% RSLogix 500 project C8011 TOPCOAT A 20170522 CBP.RSS, saved by version 8.30.00.16 %
PROJECT "C8011"    % processor: MicroLogix 1400; MAIN_PROG %

PROGRAM FILES
  LAD 2 "MAIN_PROG"  16 rungs
  LAD 3 "XFR 4"  40 rungs
  LAD 4 "XFR 5"  10 rungs
  LAD 5 "XFR 6"  10 rungs
  LAD 6 "XFR 7"  24 rungs
  LAD 7 "XFR 8"  19 rungs
  LAD 8 "XFR 9"  16 rungs
  LAD 9 "XFR 10"  27 rungs
  LAD 10 "XFR 14"  3 rungs
  LAD 11 "RFID SB"  8 rungs
  LAD 12 "Z24_Z21"  10 rungs
  LAD 13 "Z90_Z92"  4 rungs
  LAD 14 "Z49_Z54"  1 rungs
  LAD 15 "COMM"  19 rungs
  LAD 16 "XFR 69"  14 rungs

DATA FILES
  O0 OUTPUT  10 elements
  I1 INPUT  11 elements
  S2 STATUS  66 elements
  B3 BINARY  20 elements
  T4 TIMER  100 elements
  C5 COUNTER  20 elements
  R6 CONTROL  10 elements
  N7 INTEGER  100 elements
  F8 FLOAT  1 elements
  MG9   10 elements
  RI10   10 elements
  ST12 MATERIALS  50 elements
  ST13 RFID DATA  2 elements

LADDER 2 "MAIN_PROG"
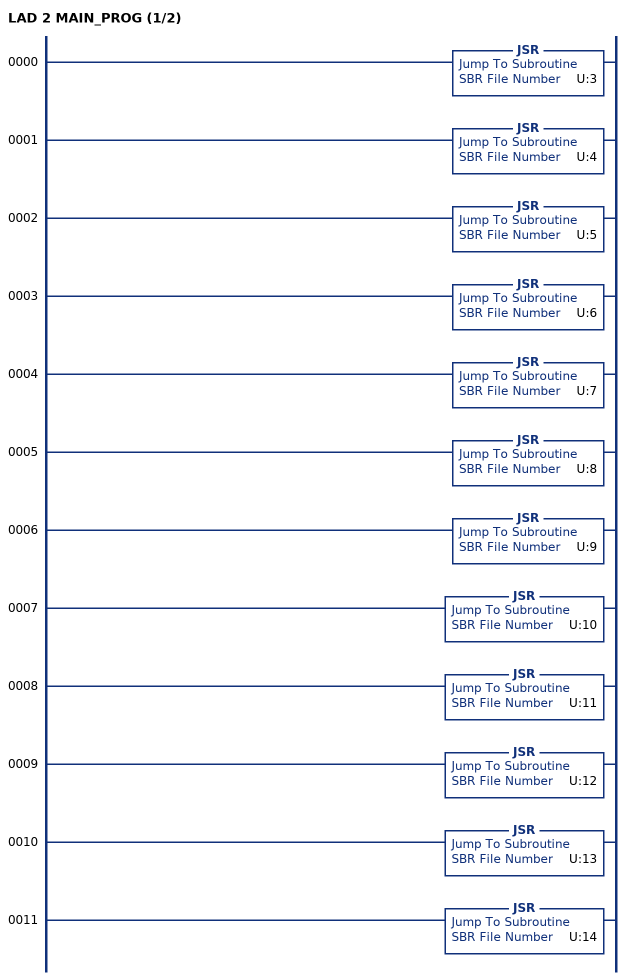
% Rung: 0 %
SOR JSR U:3 EOR
% Rung: 1 %
SOR JSR U:4 EOR
% Rung: 2 %
SOR JSR U:5 EOR
% Rung: 3 %
SOR JSR U:6 EOR
% Rung: 4 %
SOR JSR U:7 EOR
% Rung: 5 %
SOR JSR U:8 EOR
% Rung: 6 %
SOR JSR U:9 EOR
% Rung: 7 %
SOR JSR U:10 EOR
% Rung: 8 %
SOR JSR U:11 EOR
% Rung: 9 %
SOR JSR U:12 EOR
% Rung: 10 %
SOR JSR U:13 EOR
% Rung: 11 %
SOR JSR U:14 EOR

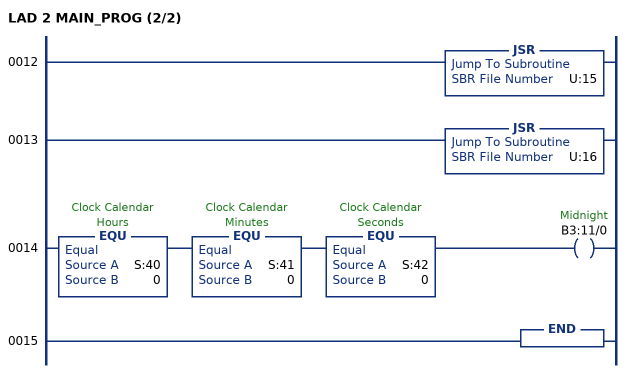
% Rung: 12 %
SOR JSR U:15 EOR
% Rung: 13 %
SOR JSR U:16 EOR
% Rung: 14 %
SOR EQU S:40 0 EQU S:41 0 EQU S:42 0 OTE B3:11/0 EOR
%   S:40  "Clock Calendar Hours" %
%   S:41  "Clock Calendar Minutes" %
%   S:42  "Clock Calendar Seconds" %
%   B3:11/0  "Midnight" %
% Rung: 15 %
SOR END EOR

LADDER 3 "XFR 4"
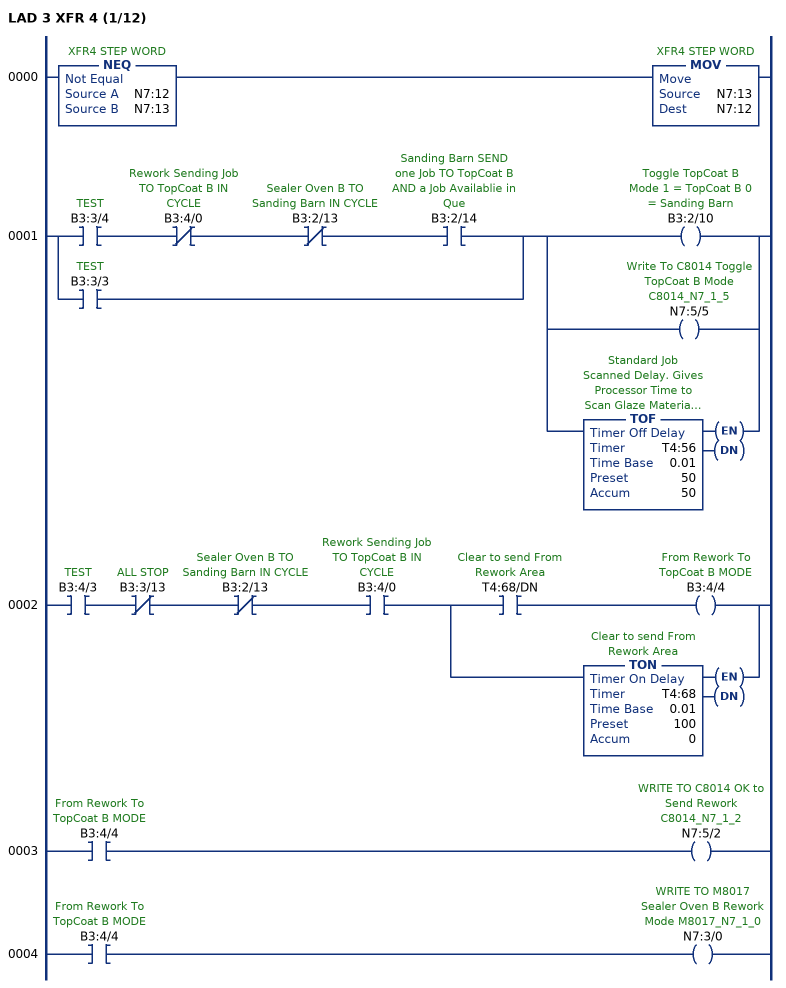
% Rung: 0 %
SOR NEQ N7:12 N7:13 MOV N7:13 N7:12 EOR
%   N7:12  "XFR4 STEP WORD" %
% Rung: 1 %
SOR BST XIC B3:3/4 XIO B3:4/0 XIO B3:2/13 XIC B3:2/14 NXB XIC B3:3/3 BND BST OTE B3:2/10 NXB OTE N7:5/5 NXB TOF T4:56 0.01 50 50 BND EOR
%   B3:3/4  "TEST" %
%   B3:4/0  "Rework Sending Job TO TopCoat B IN CYCLE" %
%   B3:2/13  "Sealer Oven B TO Sanding Barn IN CYCLE" %
%   B3:2/14  "Sanding Barn SEND one Job TO TopCoat B AND a Job Availablie in Que" %
%   B3:3/3  "TEST" %
%   B3:2/10  "Toggle TopCoat B Mode 1 = TopCoat B 0 = Sanding Barn" %
%   N7:5/5  C8014_N7_1_5  "Write To C8014 Toggle TopCoat B Mode" %
%   T4:56  "Standard Job Scanned Delay. Gives Processor Time to Scan Glaze Material Numbers" %
% Rung: 2 %
SOR XIC B3:4/3 XIO B3:3/13 XIO B3:2/13 XIC B3:4/0 BST XIC T4:68/DN OTE B3:4/4 NXB TON T4:68 0.01 100 0 BND EOR
%   B3:4/3  "TEST" %
%   B3:3/13  "ALL STOP" %
%   B3:2/13  "Sealer Oven B TO Sanding Barn IN CYCLE" %
%   B3:4/0  "Rework Sending Job TO TopCoat B IN CYCLE" %
%   T4:68  "Clear to send From Rework Area" %
%   B3:4/4  "From Rework To TopCoat B MODE" %
% Rung: 3 %
SOR XIC B3:4/4 OTE N7:5/2 EOR
%   B3:4/4  "From Rework To TopCoat B MODE" %
%   N7:5/2  C8014_N7_1_2  "WRITE TO C8014 OK to Send Rework" %
% Rung: 4 %
SOR XIC B3:4/4 OTE N7:3/0 EOR
%   B3:4/4  "From Rework To TopCoat B MODE" %
%   N7:3/0  M8017_N7_1_0  "WRITE TO M8017 Sealer Oven B Rework Mode" %

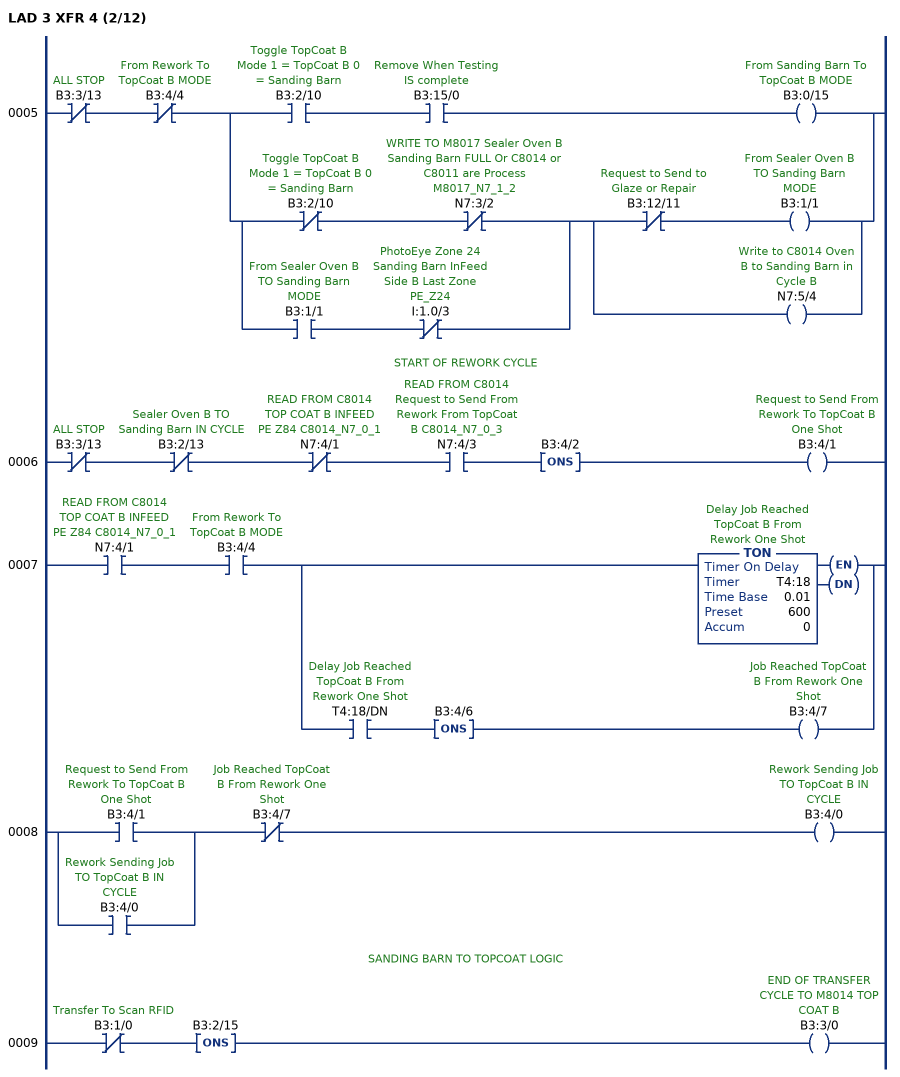
% Rung: 5 %
SOR XIO B3:3/13 XIO B3:4/4 BST XIC B3:2/10 XIC B3:15/0 OTE B3:0/15 NXB BST XIO B3:2/10 XIO N7:3/2 NXB XIC B3:1/1 XIO I:1.0/3 BND BST XIO B3:12/11 OTE B3:1/1 NXB OTE N7:5/4 BND BND EOR
%   B3:3/13  "ALL STOP" %
%   B3:4/4  "From Rework To TopCoat B MODE" %
%   B3:2/10  "Toggle TopCoat B Mode 1 = TopCoat B 0 = Sanding Barn" %
%   B3:15/0  "Remove When Testing IS complete" %
%   B3:0/15  "From Sanding Barn To TopCoat B MODE" %
%   N7:3/2  M8017_N7_1_2  "WRITE TO M8017 Sealer Oven B Sanding Barn FULL Or C8014 or C8011 are Process" %
%   B3:1/1  "From Sealer Oven B TO Sanding Barn MODE" %
%   I:1.0/3  PE_Z24  "PhotoEye Zone 24 Sanding Barn InFeed Side B Last Zone" %
%   B3:12/11  "Request to Send to Glaze or Repair" %
%   N7:5/4  B  "Write to C8014 Oven B to Sanding Barn in Cycle" %
% Rung: 6 %
% START OF REWORK CYCLE %
SOR XIO B3:3/13 XIO B3:2/13 XIO N7:4/1 XIC N7:4/3 ONS B3:4/2 OTE B3:4/1 EOR
%   B3:3/13  "ALL STOP" %
%   B3:2/13  "Sealer Oven B TO Sanding Barn IN CYCLE" %
%   N7:4/1  C8014_N7_0_1  "READ FROM C8014 TOP COAT B INFEED PE Z84" %
%   N7:4/3  C8014_N7_0_3  "READ FROM C8014 Request to Send From Rework From TopCoat B" %
%   B3:4/1  "Request to Send From Rework To TopCoat B One Shot" %
% Rung: 7 %
SOR XIC N7:4/1 XIC B3:4/4 BST TON T4:18 0.01 600 0 NXB XIC T4:18/DN ONS B3:4/6 OTE B3:4/7 BND EOR
%   N7:4/1  C8014_N7_0_1  "READ FROM C8014 TOP COAT B INFEED PE Z84" %
%   B3:4/4  "From Rework To TopCoat B MODE" %
%   T4:18  "Delay Job Reached TopCoat B From Rework One Shot" %
%   B3:4/7  "Job Reached TopCoat B From Rework One Shot" %
% Rung: 8 %
SOR BST XIC B3:4/1 NXB XIC B3:4/0 BND XIO B3:4/7 OTE B3:4/0 EOR
%   B3:4/1  "Request to Send From Rework To TopCoat B One Shot" %
%   B3:4/0  "Rework Sending Job TO TopCoat B IN CYCLE" %
%   B3:4/7  "Job Reached TopCoat B From Rework One Shot" %
% Rung: 9 %
% SANDING BARN TO TOPCOAT LOGIC %
SOR XIO B3:1/0 ONS B3:2/15 OTE B3:3/0 EOR
%   B3:1/0  "Transfer To Scan RFID" %
%   B3:3/0  "END OF TRANSFER CYCLE TO M8014 TOP COAT B" %

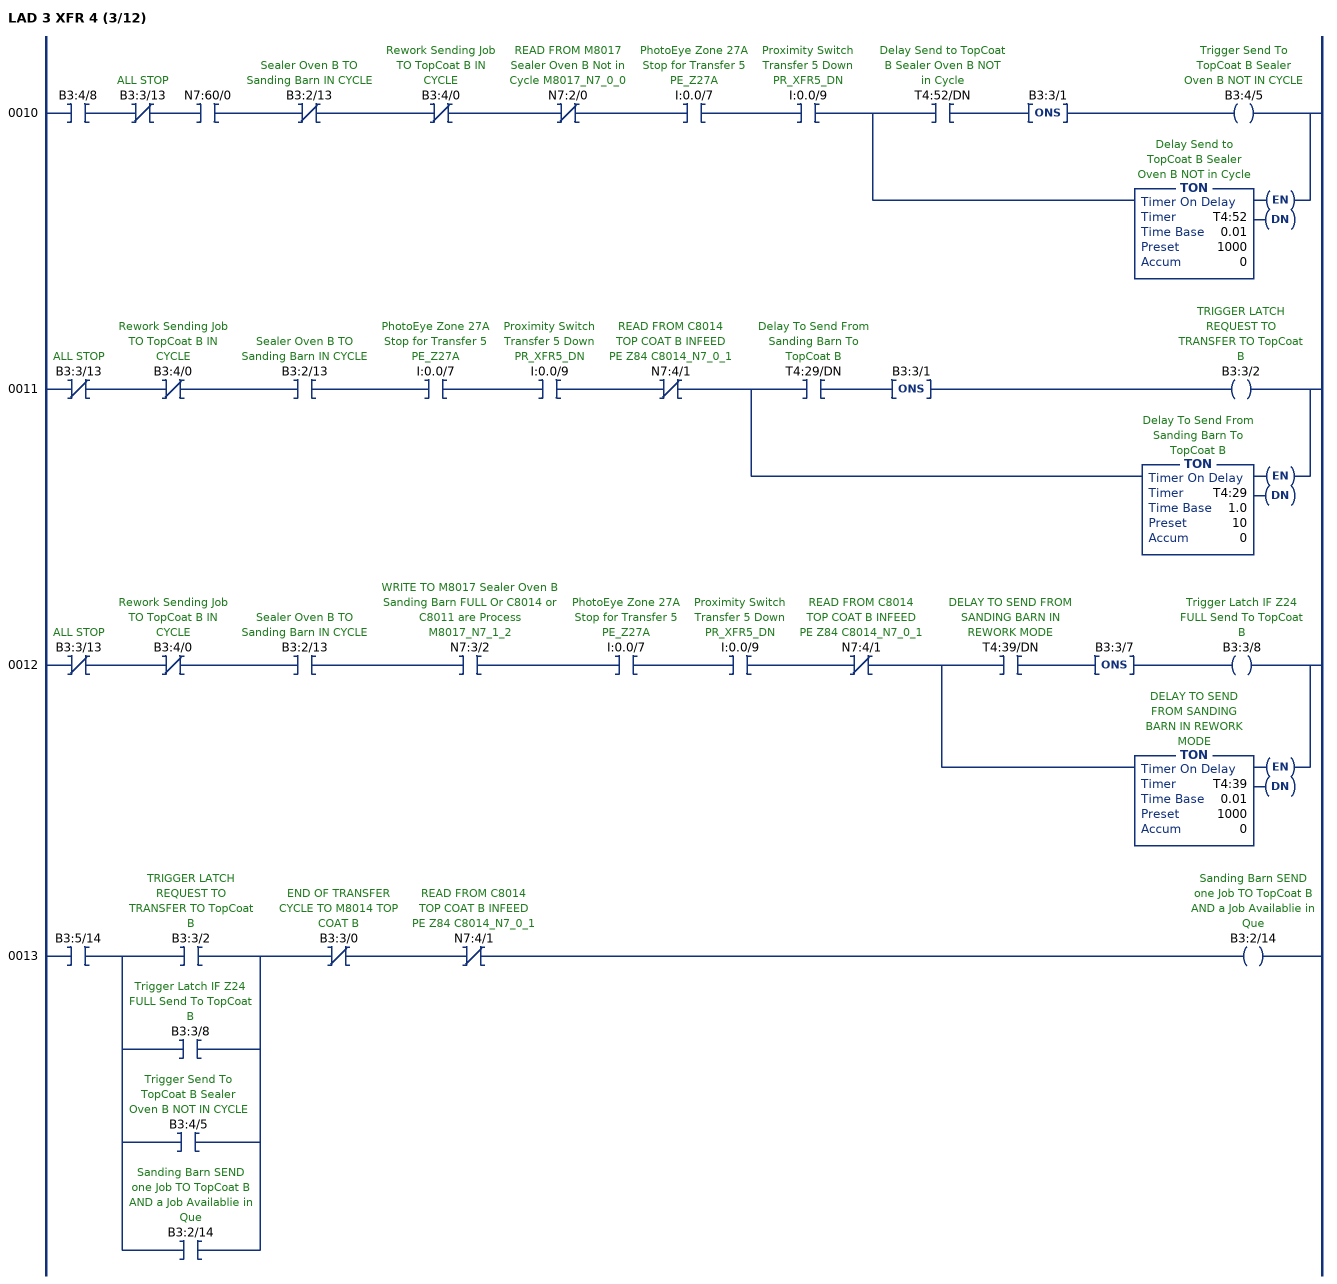
% Rung: 10 %
SOR XIC B3:4/8 XIO B3:3/13 XIC N7:60/0 XIO B3:2/13 XIO B3:4/0 XIO N7:2/0 XIC I:0.0/7 XIC I:0.0/9 BST XIC T4:52/DN ONS B3:3/1 OTE B3:4/5 NXB TON T4:52 0.01 1000 0 BND EOR
%   B3:3/13  "ALL STOP" %
%   B3:2/13  "Sealer Oven B TO Sanding Barn IN CYCLE" %
%   B3:4/0  "Rework Sending Job TO TopCoat B IN CYCLE" %
%   N7:2/0  M8017_N7_0_0  "READ FROM M8017 Sealer Oven B Not in Cycle" %
%   I:0.0/7  PE_Z27A  "PhotoEye Zone 27A Stop for Transfer 5" %
%   I:0.0/9  PR_XFR5_DN  "Proximity Switch Transfer 5 Down" %
%   T4:52  "Delay Send to TopCoat B Sealer Oven B NOT in Cycle" %
%   B3:4/5  "Trigger Send To TopCoat B Sealer Oven B NOT IN CYCLE" %
% Rung: 11 %
SOR XIO B3:3/13 XIO B3:4/0 XIC B3:2/13 XIC I:0.0/7 XIC I:0.0/9 XIO N7:4/1 BST XIC T4:29/DN ONS B3:3/1 OTE B3:3/2 NXB TON T4:29 1.0 10 0 BND EOR
%   B3:3/13  "ALL STOP" %
%   B3:4/0  "Rework Sending Job TO TopCoat B IN CYCLE" %
%   B3:2/13  "Sealer Oven B TO Sanding Barn IN CYCLE" %
%   I:0.0/7  PE_Z27A  "PhotoEye Zone 27A Stop for Transfer 5" %
%   I:0.0/9  PR_XFR5_DN  "Proximity Switch Transfer 5 Down" %
%   N7:4/1  C8014_N7_0_1  "READ FROM C8014 TOP COAT B INFEED PE Z84" %
%   T4:29  "Delay To Send From Sanding Barn To TopCoat B" %
%   B3:3/2  "TRIGGER LATCH REQUEST TO TRANSFER TO TopCoat B" %
% Rung: 12 %
SOR XIO B3:3/13 XIO B3:4/0 XIC B3:2/13 XIC N7:3/2 XIC I:0.0/7 XIC I:0.0/9 XIO N7:4/1 BST XIC T4:39/DN ONS B3:3/7 OTE B3:3/8 NXB TON T4:39 0.01 1000 0 BND EOR
%   B3:3/13  "ALL STOP" %
%   B3:4/0  "Rework Sending Job TO TopCoat B IN CYCLE" %
%   B3:2/13  "Sealer Oven B TO Sanding Barn IN CYCLE" %
%   N7:3/2  M8017_N7_1_2  "WRITE TO M8017 Sealer Oven B Sanding Barn FULL Or C8014 or C8011 are Process" %
%   I:0.0/7  PE_Z27A  "PhotoEye Zone 27A Stop for Transfer 5" %
%   I:0.0/9  PR_XFR5_DN  "Proximity Switch Transfer 5 Down" %
%   N7:4/1  C8014_N7_0_1  "READ FROM C8014 TOP COAT B INFEED PE Z84" %
%   T4:39  "DELAY TO SEND FROM SANDING BARN IN REWORK MODE" %
%   B3:3/8  "Trigger Latch IF Z24 FULL Send To TopCoat B" %
% Rung: 13 %
SOR XIC B3:5/14 BST XIC B3:3/2 NXB XIC B3:3/8 NXB XIC B3:4/5 NXB XIC B3:2/14 BND XIO B3:3/0 XIO N7:4/1 OTE B3:2/14 EOR
%   B3:3/2  "TRIGGER LATCH REQUEST TO TRANSFER TO TopCoat B" %
%   B3:3/8  "Trigger Latch IF Z24 FULL Send To TopCoat B" %
%   B3:4/5  "Trigger Send To TopCoat B Sealer Oven B NOT IN CYCLE" %
%   B3:2/14  "Sanding Barn SEND one Job TO TopCoat B AND a Job Availablie in Que" %
%   B3:3/0  "END OF TRANSFER CYCLE TO M8014 TOP COAT B" %
%   N7:4/1  C8014_N7_0_1  "READ FROM C8014 TOP COAT B INFEED PE Z84" %

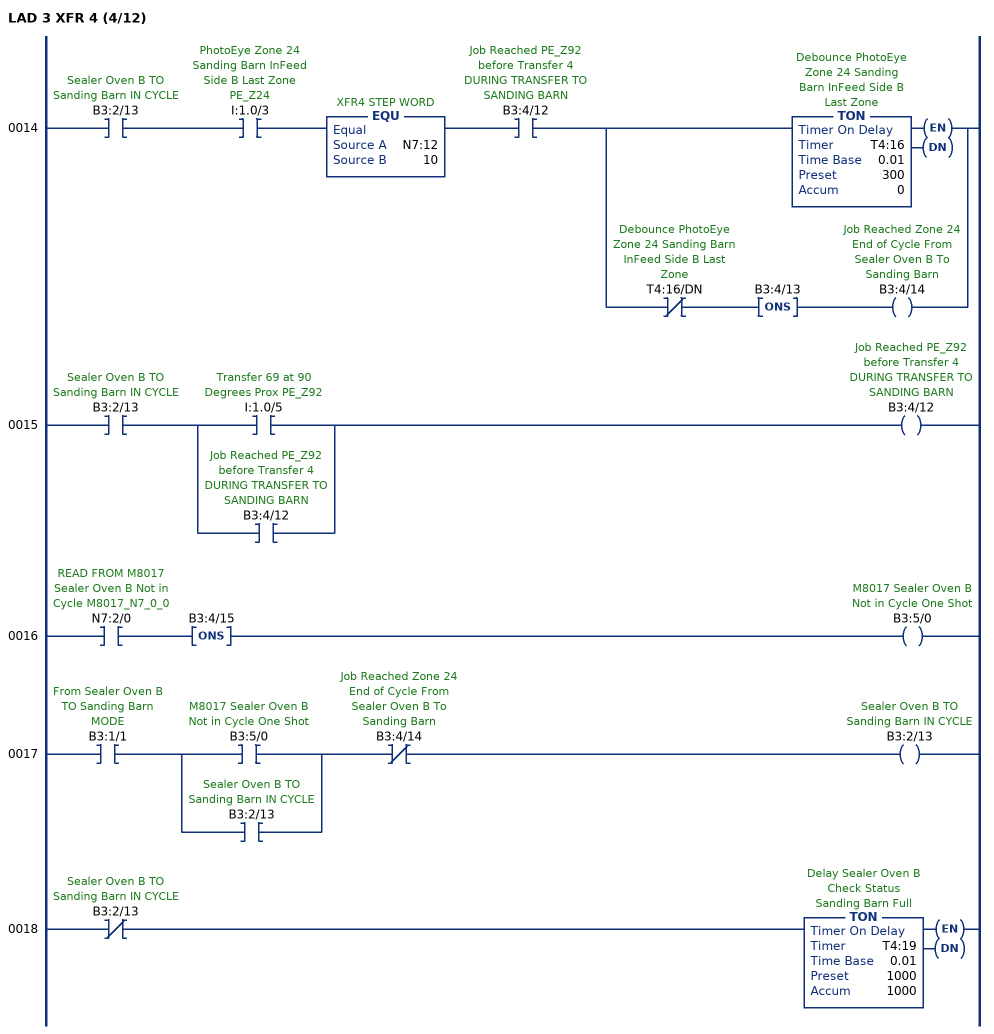
% Rung: 14 %
SOR XIC B3:2/13 XIC I:1.0/3 EQU N7:12 10 XIC B3:4/12 BST TON T4:16 0.01 300 0 NXB XIO T4:16/DN ONS B3:4/13 OTE B3:4/14 BND EOR
%   B3:2/13  "Sealer Oven B TO Sanding Barn IN CYCLE" %
%   I:1.0/3  PE_Z24  "PhotoEye Zone 24 Sanding Barn InFeed Side B Last Zone" %
%   N7:12  "XFR4 STEP WORD" %
%   B3:4/12  "Job Reached PE_Z92 before Transfer 4 DURING TRANSFER TO SANDING BARN" %
%   T4:16  "Debounce PhotoEye Zone 24 Sanding Barn InFeed Side B Last Zone" %
%   B3:4/14  "Job Reached Zone 24 End of Cycle From Sealer Oven B To Sanding Barn" %
% Rung: 15 %
SOR XIC B3:2/13 BST XIC I:1.0/5 NXB XIC B3:4/12 BND OTE B3:4/12 EOR
%   B3:2/13  "Sealer Oven B TO Sanding Barn IN CYCLE" %
%   I:1.0/5  PE_Z92  "Transfer 69 at 90 Degrees Prox" %
%   B3:4/12  "Job Reached PE_Z92 before Transfer 4 DURING TRANSFER TO SANDING BARN" %
% Rung: 16 %
SOR XIC N7:2/0 ONS B3:4/15 OTE B3:5/0 EOR
%   N7:2/0  M8017_N7_0_0  "READ FROM M8017 Sealer Oven B Not in Cycle" %
%   B3:5/0  "M8017 Sealer Oven B Not in Cycle One Shot" %
% Rung: 17 %
SOR XIC B3:1/1 BST XIC B3:5/0 NXB XIC B3:2/13 BND XIO B3:4/14 OTE B3:2/13 EOR
%   B3:1/1  "From Sealer Oven B TO Sanding Barn MODE" %
%   B3:5/0  "M8017 Sealer Oven B Not in Cycle One Shot" %
%   B3:2/13  "Sealer Oven B TO Sanding Barn IN CYCLE" %
%   B3:4/14  "Job Reached Zone 24 End of Cycle From Sealer Oven B To Sanding Barn" %
% Rung: 18 %
SOR XIO B3:2/13 TON T4:19 0.01 1000 1000 EOR
%   B3:2/13  "Sealer Oven B TO Sanding Barn IN CYCLE" %
%   T4:19  "Delay Sealer Oven B Check Status Sanding Barn Full" %

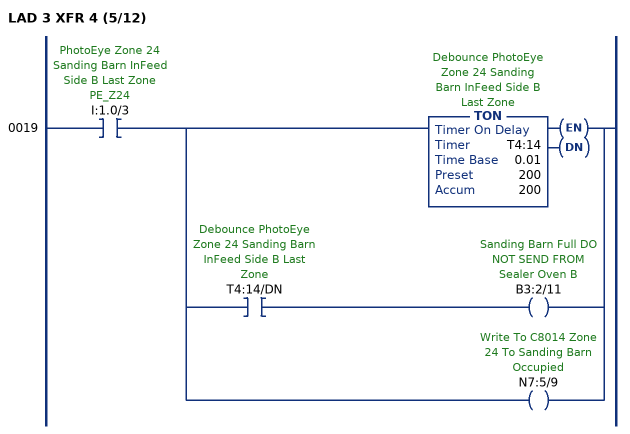
% Rung: 19 %
SOR XIC I:1.0/3 BST TON T4:14 0.01 200 200 NXB XIC T4:14/DN OTE B3:2/11 NXB OTE N7:5/9 BND EOR
%   I:1.0/3  PE_Z24  "PhotoEye Zone 24 Sanding Barn InFeed Side B Last Zone" %
%   T4:14  "Debounce PhotoEye Zone 24 Sanding Barn InFeed Side B Last Zone" %
%   B3:2/11  "Sanding Barn Full DO NOT SEND FROM Sealer Oven B" %
%   N7:5/9  "Write To C8014 Zone 24 To Sanding Barn Occupied" %

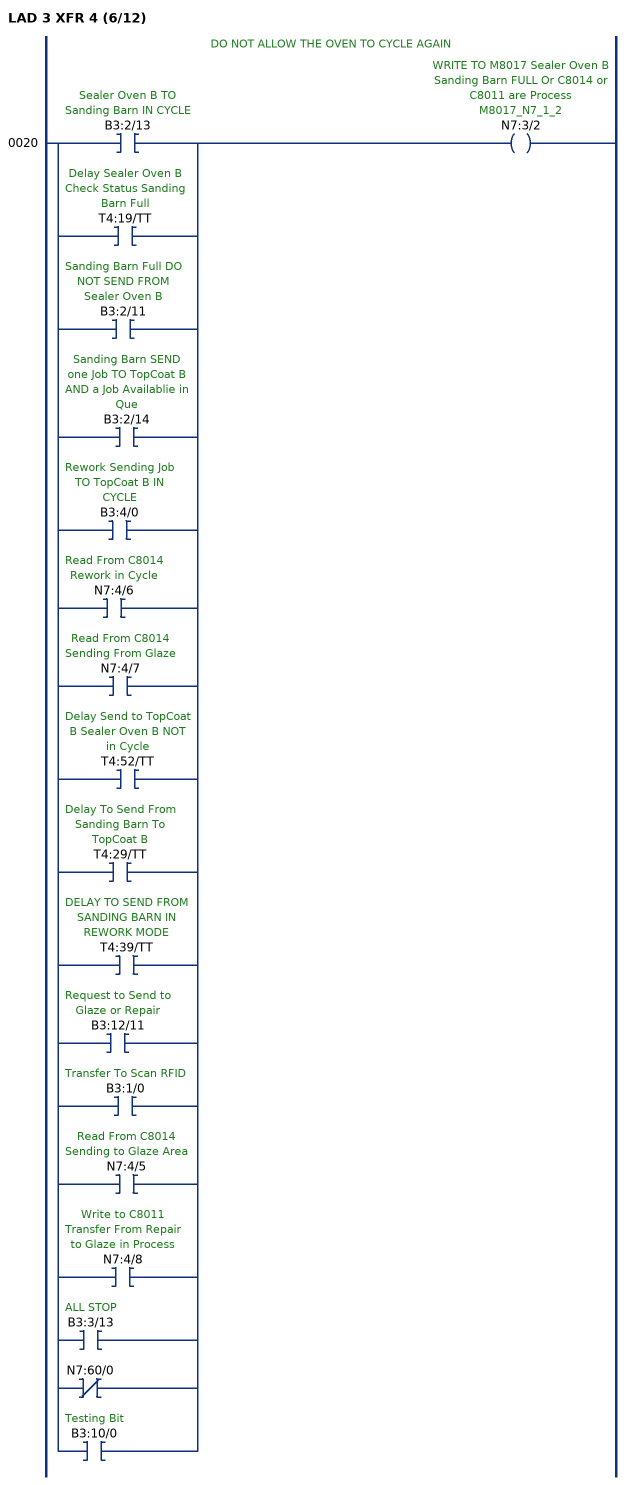
% Rung: 20 %
% DO NOT ALLOW THE OVEN TO CYCLE AGAIN %
SOR BST XIC B3:2/13 NXB XIC T4:19/TT NXB XIC B3:2/11 NXB XIC B3:2/14 NXB XIC B3:4/0 NXB XIC N7:4/6 NXB XIC N7:4/7 NXB XIC T4:52/TT NXB XIC T4:29/TT NXB XIC T4:39/TT NXB XIC B3:12/11 NXB XIC B3:1/0 NXB XIC N7:4/5 NXB XIC N7:4/8 NXB XIC B3:3/13 NXB XIO N7:60/0 NXB XIC B3:10/0 BND OTE N7:3/2 EOR
%   B3:2/13  "Sealer Oven B TO Sanding Barn IN CYCLE" %
%   T4:19  "Delay Sealer Oven B Check Status Sanding Barn Full" %
%   B3:2/11  "Sanding Barn Full DO NOT SEND FROM Sealer Oven B" %
%   B3:2/14  "Sanding Barn SEND one Job TO TopCoat B AND a Job Availablie in Que" %
%   B3:4/0  "Rework Sending Job TO TopCoat B IN CYCLE" %
%   N7:4/6  "Read From C8014 Rework in Cycle" %
%   N7:4/7  "Read From C8014 Sending From Glaze" %
%   T4:52  "Delay Send to TopCoat B Sealer Oven B NOT in Cycle" %
%   T4:29  "Delay To Send From Sanding Barn To TopCoat B" %
%   T4:39  "DELAY TO SEND FROM SANDING BARN IN REWORK MODE" %
%   B3:12/11  "Request to Send to Glaze or Repair" %
%   B3:1/0  "Transfer To Scan RFID" %
%   N7:4/5  "Read From C8014 Sending to Glaze Area" %
%   N7:4/8  "Write to C8011 Transfer From Repair to Glaze in Process" %
%   B3:3/13  "ALL STOP" %
%   B3:10/0  "Testing Bit" %
%   N7:3/2  M8017_N7_1_2  "WRITE TO M8017 Sealer Oven B Sanding Barn FULL Or C8014 or C8011 are Process" %

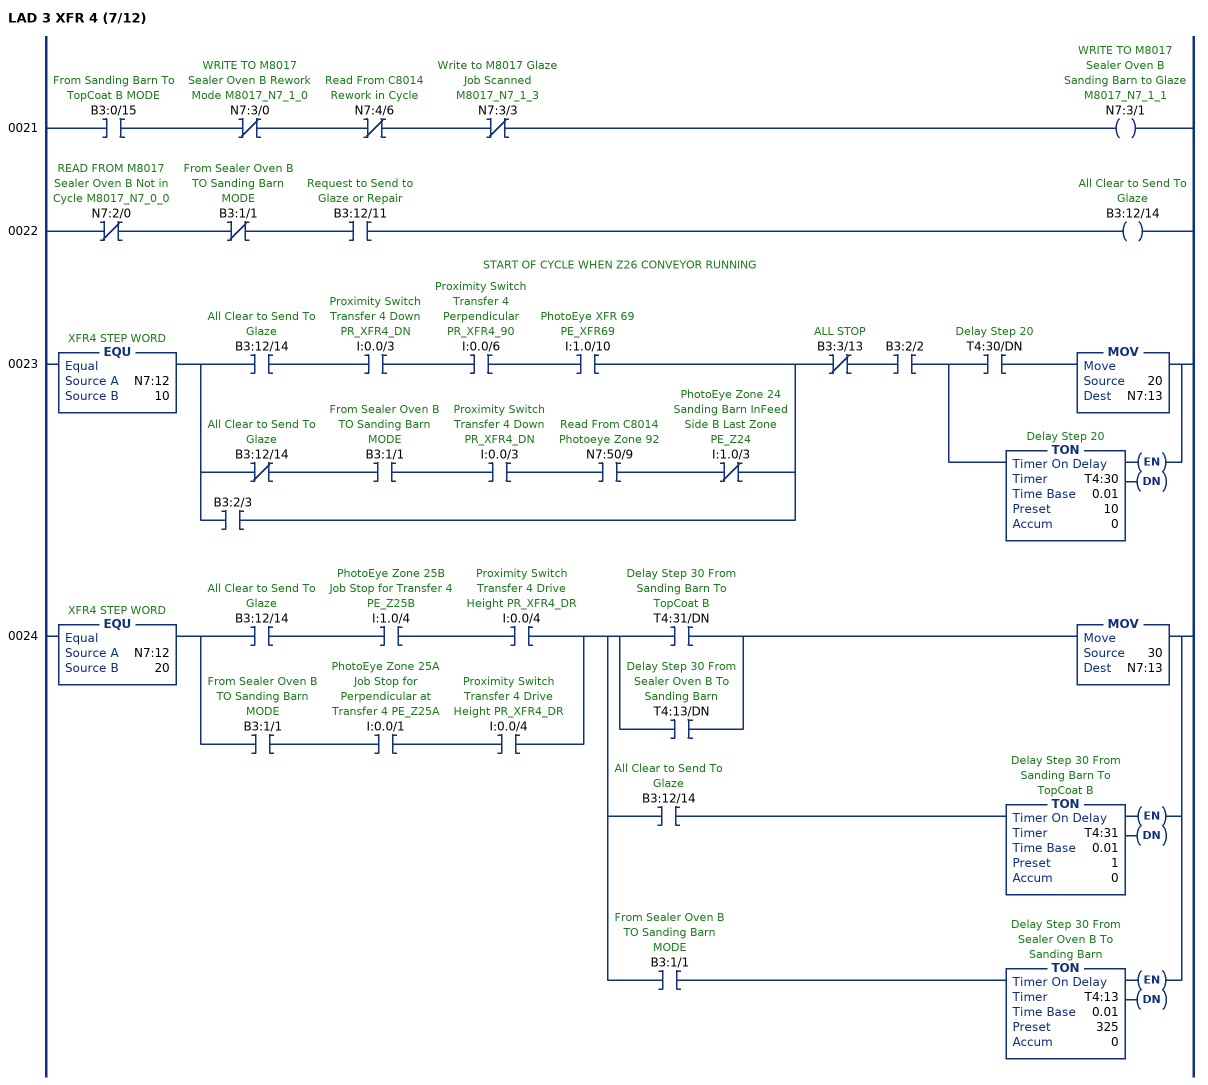
% Rung: 21 %
SOR XIC B3:0/15 XIO N7:3/0 XIO N7:4/6 XIO N7:3/3 OTE N7:3/1 EOR
%   B3:0/15  "From Sanding Barn To TopCoat B MODE" %
%   N7:3/0  M8017_N7_1_0  "WRITE TO M8017 Sealer Oven B Rework Mode" %
%   N7:4/6  "Read From C8014 Rework in Cycle" %
%   N7:3/3  M8017_N7_1_3  "Write to M8017 Glaze Job Scanned" %
%   N7:3/1  M8017_N7_1_1  "WRITE TO M8017 Sealer Oven B Sanding Barn to Glaze" %
% Rung: 22 %
SOR XIO N7:2/0 XIO B3:1/1 XIC B3:12/11 OTE B3:12/14 EOR
%   N7:2/0  M8017_N7_0_0  "READ FROM M8017 Sealer Oven B Not in Cycle" %
%   B3:1/1  "From Sealer Oven B TO Sanding Barn MODE" %
%   B3:12/11  "Request to Send to Glaze or Repair" %
%   B3:12/14  "All Clear to Send To Glaze" %
% Rung: 23 %
% START OF CYCLE WHEN Z26 CONVEYOR RUNNING %
SOR EQU N7:12 10 BST XIC B3:12/14 XIC I:0.0/3 XIC I:0.0/6 XIC I:1.0/10 NXB XIO B3:12/14 XIC B3:1/1 XIC I:0.0/3 XIC N7:50/9 XIO I:1.0/3 NXB XIC B3:2/3 BND XIO B3:3/13 XIC B3:2/2 BST XIC T4:30/DN MOV 20 N7:13 NXB TON T4:30 0.01 10 0 BND EOR
%   N7:12  "XFR4 STEP WORD" %
%   B3:12/14  "All Clear to Send To Glaze" %
%   I:0.0/3  PR_XFR4_DN  "Proximity Switch Transfer 4 Down" %
%   I:0.0/6  PR_XFR4_90  "Proximity Switch Transfer 4 Perpendicular" %
%   I:1.0/10  PE_XFR69  "PhotoEye XFR 69" %
%   B3:1/1  "From Sealer Oven B TO Sanding Barn MODE" %
%   N7:50/9  "Read From C8014 Photoeye Zone 92" %
%   I:1.0/3  PE_Z24  "PhotoEye Zone 24 Sanding Barn InFeed Side B Last Zone" %
%   B3:3/13  "ALL STOP" %
%   T4:30  "Delay Step 20" %
% Rung: 24 %
SOR EQU N7:12 20 BST XIC B3:12/14 XIC I:1.0/4 XIC I:0.0/4 NXB XIC B3:1/1 XIC I:0.0/1 XIC I:0.0/4 BND BST BST XIC T4:31/DN NXB XIC T4:13/DN BND MOV 30 N7:13 NXB XIC B3:12/14 TON T4:31 0.01 1 0 NXB XIC B3:1/1 TON T4:13 0.01 325 0 BND EOR
%   N7:12  "XFR4 STEP WORD" %
%   B3:12/14  "All Clear to Send To Glaze" %
%   I:1.0/4  PE_Z25B  "PhotoEye Zone 25B Job Stop for Transfer 4" %
%   I:0.0/4  PR_XFR4_DR  "Proximity Switch Transfer 4 Drive Height" %
%   B3:1/1  "From Sealer Oven B TO Sanding Barn MODE" %
%   I:0.0/1  PE_Z25A  "PhotoEye Zone 25A Job Stop for Perpendicular at Transfer 4" %
%   T4:31  "Delay Step 30 From Sanding Barn To TopCoat B" %
%   T4:13  "Delay Step 30 From Sealer Oven B To Sanding Barn" %

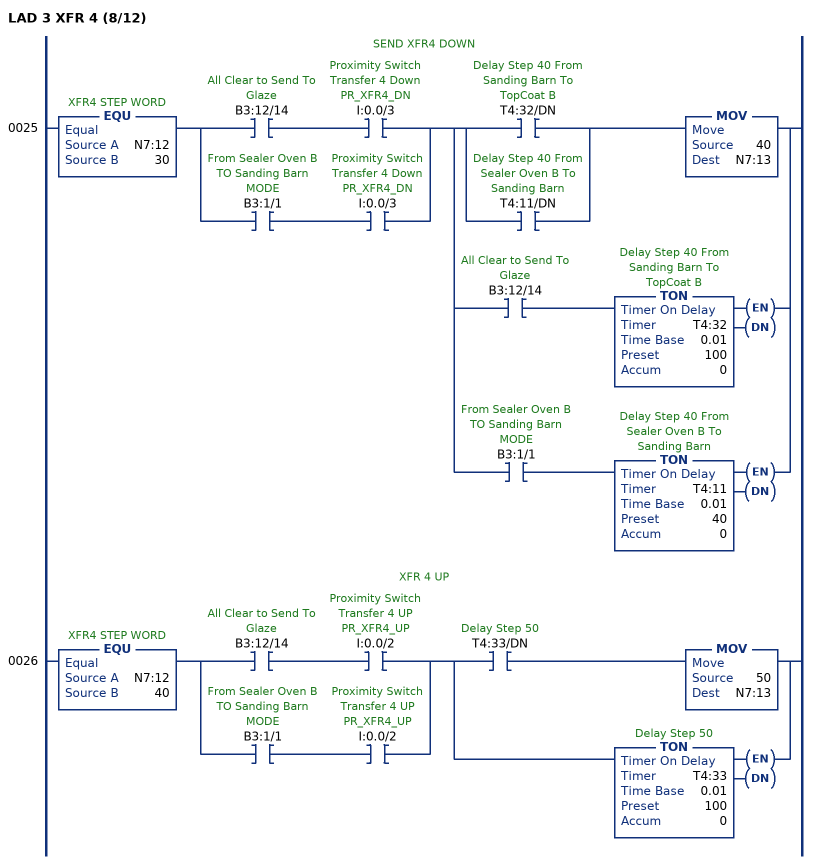
% Rung: 25 %
% SEND XFR4 DOWN %
SOR EQU N7:12 30 BST XIC B3:12/14 XIC I:0.0/3 NXB XIC B3:1/1 XIC I:0.0/3 BND BST BST XIC T4:32/DN NXB XIC T4:11/DN BND MOV 40 N7:13 NXB XIC B3:12/14 TON T4:32 0.01 100 0 NXB XIC B3:1/1 TON T4:11 0.01 40 0 BND EOR
%   N7:12  "XFR4 STEP WORD" %
%   B3:12/14  "All Clear to Send To Glaze" %
%   I:0.0/3  PR_XFR4_DN  "Proximity Switch Transfer 4 Down" %
%   B3:1/1  "From Sealer Oven B TO Sanding Barn MODE" %
%   T4:32  "Delay Step 40 From Sanding Barn To TopCoat B" %
%   T4:11  "Delay Step 40 From Sealer Oven B To Sanding Barn" %
% Rung: 26 %
% XFR 4 UP %
SOR EQU N7:12 40 BST XIC B3:12/14 XIC I:0.0/2 NXB XIC B3:1/1 XIC I:0.0/2 BND BST XIC T4:33/DN MOV 50 N7:13 NXB TON T4:33 0.01 100 0 BND EOR
%   N7:12  "XFR4 STEP WORD" %
%   B3:12/14  "All Clear to Send To Glaze" %
%   I:0.0/2  PR_XFR4_UP  "Proximity Switch Transfer 4 UP" %
%   B3:1/1  "From Sealer Oven B TO Sanding Barn MODE" %
%   T4:33  "Delay Step 50" %

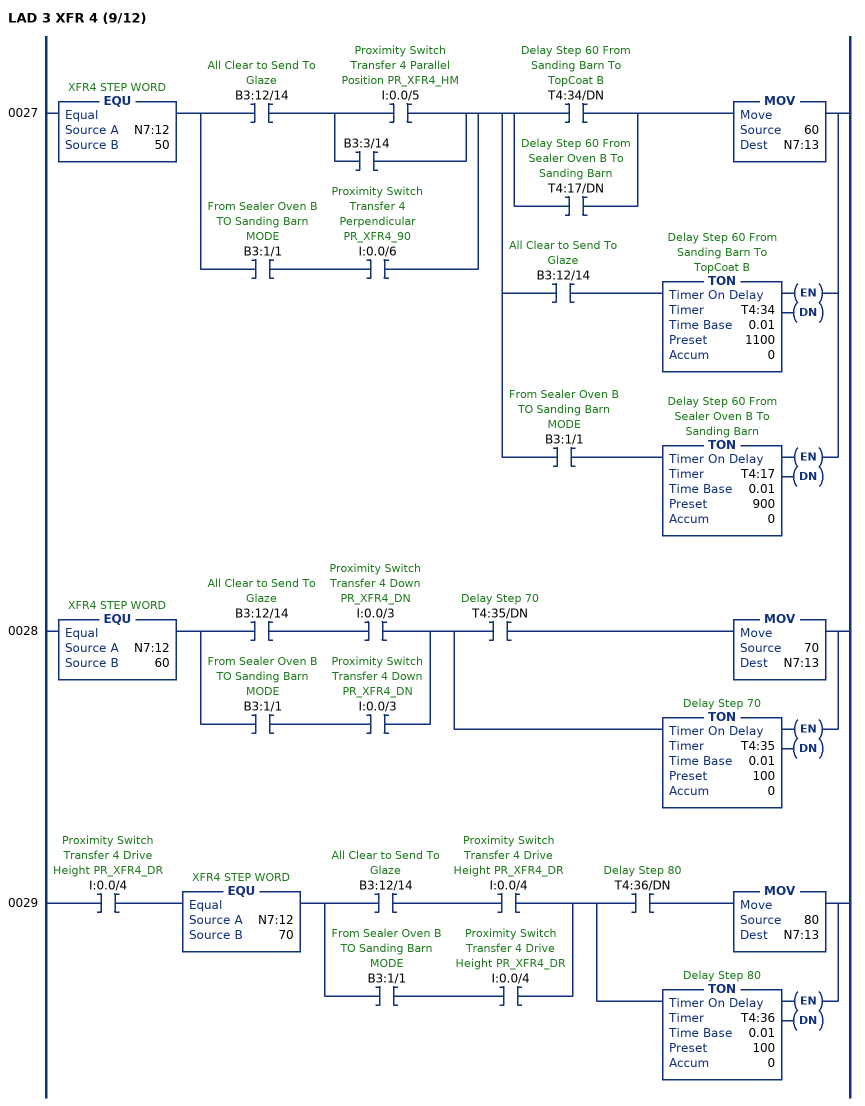
% Rung: 27 %
SOR EQU N7:12 50 BST XIC B3:12/14 BST XIC I:0.0/5 NXB XIC B3:3/14 BND NXB XIC B3:1/1 XIC I:0.0/6 BND BST BST XIC T4:34/DN NXB XIC T4:17/DN BND MOV 60 N7:13 NXB XIC B3:12/14 TON T4:34 0.01 1100 0 NXB XIC B3:1/1 TON T4:17 0.01 900 0 BND EOR
%   N7:12  "XFR4 STEP WORD" %
%   B3:12/14  "All Clear to Send To Glaze" %
%   I:0.0/5  PR_XFR4_HM  "Proximity Switch Transfer 4 Parallel Position" %
%   B3:1/1  "From Sealer Oven B TO Sanding Barn MODE" %
%   I:0.0/6  PR_XFR4_90  "Proximity Switch Transfer 4 Perpendicular" %
%   T4:34  "Delay Step 60 From Sanding Barn To TopCoat B" %
%   T4:17  "Delay Step 60 From Sealer Oven B To Sanding Barn" %
% Rung: 28 %
SOR EQU N7:12 60 BST XIC B3:12/14 XIC I:0.0/3 NXB XIC B3:1/1 XIC I:0.0/3 BND BST XIC T4:35/DN MOV 70 N7:13 NXB TON T4:35 0.01 100 0 BND EOR
%   N7:12  "XFR4 STEP WORD" %
%   B3:12/14  "All Clear to Send To Glaze" %
%   I:0.0/3  PR_XFR4_DN  "Proximity Switch Transfer 4 Down" %
%   B3:1/1  "From Sealer Oven B TO Sanding Barn MODE" %
%   T4:35  "Delay Step 70" %
% Rung: 29 %
SOR XIC I:0.0/4 EQU N7:12 70 BST XIC B3:12/14 XIC I:0.0/4 NXB XIC B3:1/1 XIC I:0.0/4 BND BST XIC T4:36/DN MOV 80 N7:13 NXB TON T4:36 0.01 100 0 BND EOR
%   I:0.0/4  PR_XFR4_DR  "Proximity Switch Transfer 4 Drive Height" %
%   N7:12  "XFR4 STEP WORD" %
%   B3:12/14  "All Clear to Send To Glaze" %
%   B3:1/1  "From Sealer Oven B TO Sanding Barn MODE" %
%   T4:36  "Delay Step 80" %

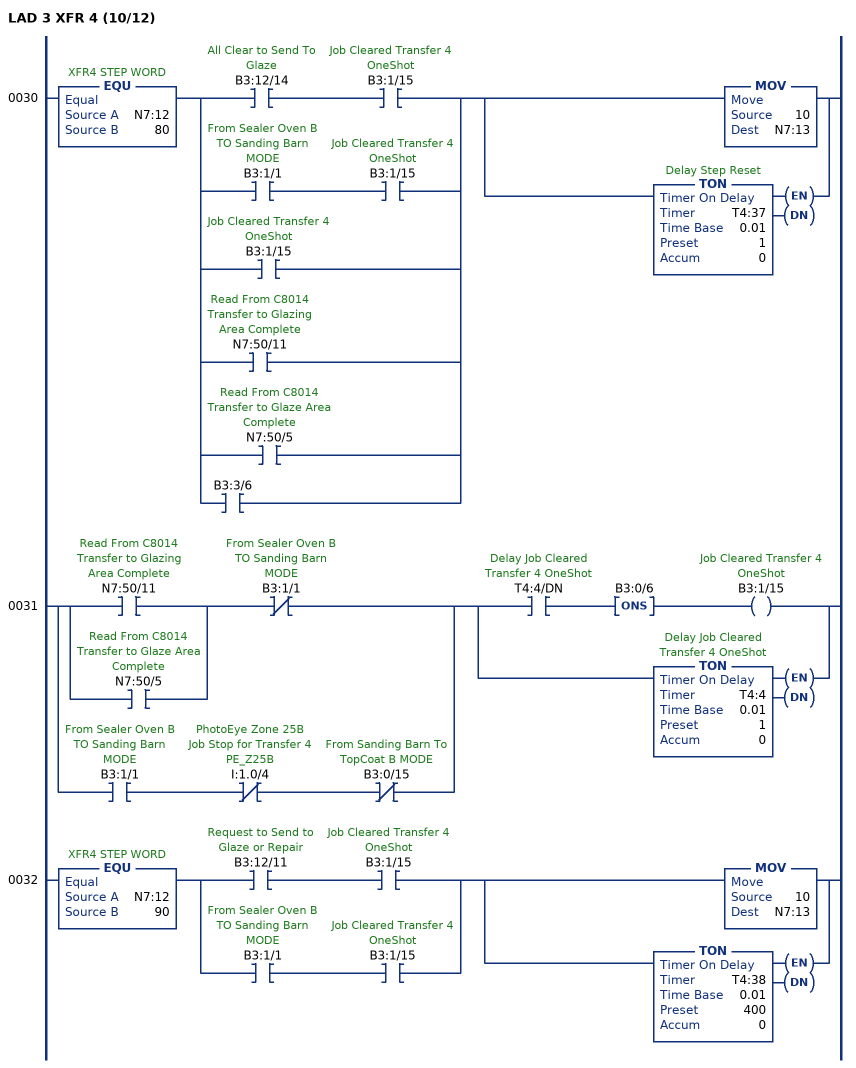
% Rung: 30 %
SOR EQU N7:12 80 BST XIC B3:12/14 XIC B3:1/15 NXB XIC B3:1/1 XIC B3:1/15 NXB XIC B3:1/15 NXB XIC N7:50/11 NXB XIC N7:50/5 NXB XIC B3:3/6 BND BST MOV 10 N7:13 NXB TON T4:37 0.01 1 0 BND EOR
%   N7:12  "XFR4 STEP WORD" %
%   B3:12/14  "All Clear to Send To Glaze" %
%   B3:1/15  "Job Cleared Transfer 4 OneShot" %
%   B3:1/1  "From Sealer Oven B TO Sanding Barn MODE" %
%   N7:50/11  "Read From C8014 Transfer to Glazing Area Complete" %
%   N7:50/5  "Read From C8014 Transfer to Glaze Area Complete" %
%   T4:37  "Delay Step Reset" %
% Rung: 31 %
SOR BST BST XIC N7:50/11 NXB XIC N7:50/5 BND XIO B3:1/1 NXB XIC B3:1/1 XIO I:1.0/4 XIO B3:0/15 BND BST XIC T4:4/DN ONS B3:0/6 OTE B3:1/15 NXB TON T4:4 0.01 1 0 BND EOR
%   N7:50/11  "Read From C8014 Transfer to Glazing Area Complete" %
%   N7:50/5  "Read From C8014 Transfer to Glaze Area Complete" %
%   B3:1/1  "From Sealer Oven B TO Sanding Barn MODE" %
%   I:1.0/4  PE_Z25B  "PhotoEye Zone 25B Job Stop for Transfer 4" %
%   B3:0/15  "From Sanding Barn To TopCoat B MODE" %
%   T4:4  "Delay Job Cleared Transfer 4 OneShot" %
%   B3:1/15  "Job Cleared Transfer 4 OneShot" %
% Rung: 32 %
SOR EQU N7:12 90 BST XIC B3:12/11 XIC B3:1/15 NXB XIC B3:1/1 XIC B3:1/15 BND BST MOV 10 N7:13 NXB TON T4:38 0.01 400 0 BND EOR
%   N7:12  "XFR4 STEP WORD" %
%   B3:12/11  "Request to Send to Glaze or Repair" %
%   B3:1/15  "Job Cleared Transfer 4 OneShot" %
%   B3:1/1  "From Sealer Oven B TO Sanding Barn MODE" %

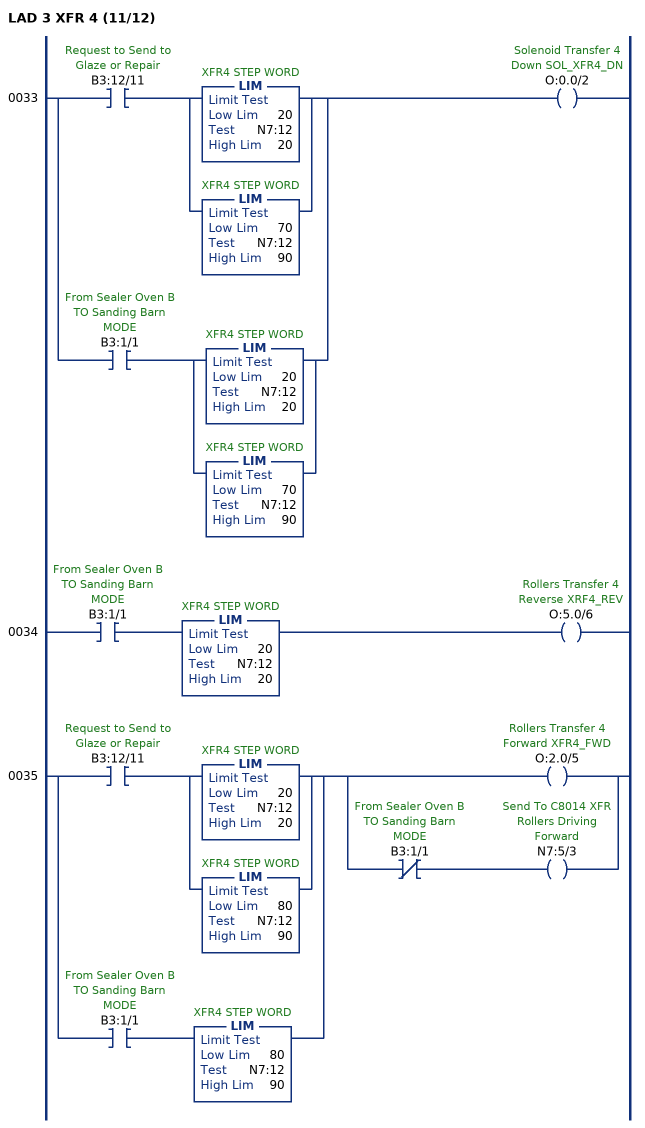
% Rung: 33 %
SOR BST XIC B3:12/11 BST LIM 20 N7:12 20 NXB LIM 70 N7:12 90 BND NXB XIC B3:1/1 BST LIM 20 N7:12 20 NXB LIM 70 N7:12 90 BND BND OTE O:0.0/2 EOR
%   B3:12/11  "Request to Send to Glaze or Repair" %
%   N7:12  "XFR4 STEP WORD" %
%   B3:1/1  "From Sealer Oven B TO Sanding Barn MODE" %
%   O:0.0/2  SOL_XFR4_DN  "Solenoid Transfer 4 Down" %
% Rung: 34 %
SOR XIC B3:1/1 LIM 20 N7:12 20 OTE O:5.0/6 EOR
%   B3:1/1  "From Sealer Oven B TO Sanding Barn MODE" %
%   N7:12  "XFR4 STEP WORD" %
%   O:5.0/6  XRF4_REV  "Rollers Transfer 4 Reverse" %
% Rung: 35 %
SOR BST XIC B3:12/11 BST LIM 20 N7:12 20 NXB LIM 80 N7:12 90 BND NXB XIC B3:1/1 LIM 80 N7:12 90 BND BST OTE O:2.0/5 NXB XIO B3:1/1 OTE N7:5/3 BND EOR
%   B3:12/11  "Request to Send to Glaze or Repair" %
%   N7:12  "XFR4 STEP WORD" %
%   B3:1/1  "From Sealer Oven B TO Sanding Barn MODE" %
%   O:2.0/5  XFR4_FWD  "Rollers Transfer 4 Forward" %
%   N7:5/3  "Send To C8014 XFR Rollers Driving Forward" %

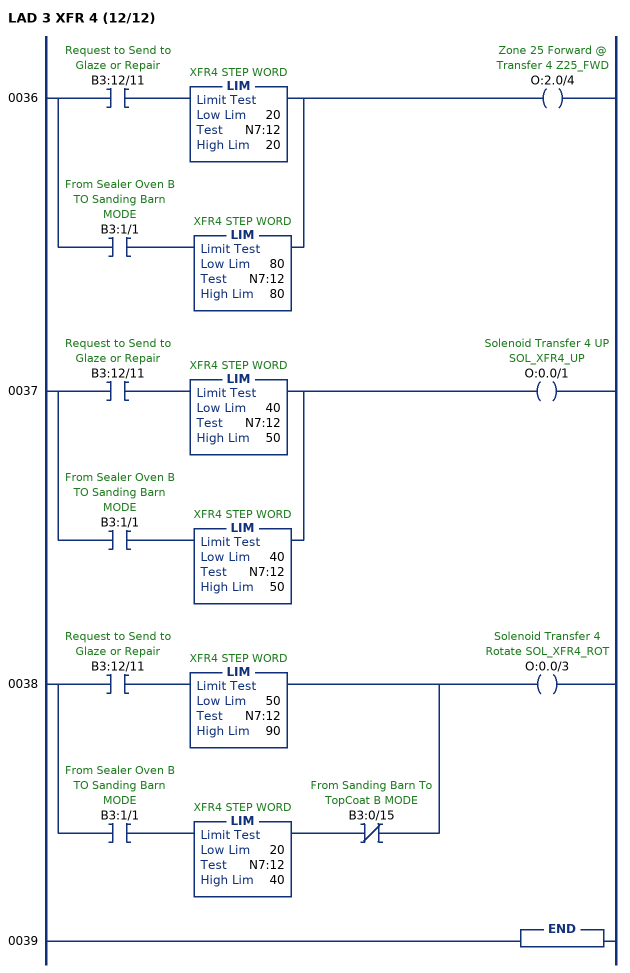
% Rung: 36 %
SOR BST XIC B3:12/11 LIM 20 N7:12 20 NXB XIC B3:1/1 LIM 80 N7:12 80 BND OTE O:2.0/4 EOR
%   B3:12/11  "Request to Send to Glaze or Repair" %
%   N7:12  "XFR4 STEP WORD" %
%   B3:1/1  "From Sealer Oven B TO Sanding Barn MODE" %
%   O:2.0/4  Z25_FWD  "Zone 25 Forward @ Transfer 4" %
% Rung: 37 %
SOR BST XIC B3:12/11 LIM 40 N7:12 50 NXB XIC B3:1/1 LIM 40 N7:12 50 BND OTE O:0.0/1 EOR
%   B3:12/11  "Request to Send to Glaze or Repair" %
%   N7:12  "XFR4 STEP WORD" %
%   B3:1/1  "From Sealer Oven B TO Sanding Barn MODE" %
%   O:0.0/1  SOL_XFR4_UP  "Solenoid Transfer 4 UP" %
% Rung: 38 %
SOR BST XIC B3:12/11 LIM 50 N7:12 90 NXB XIC B3:1/1 LIM 20 N7:12 40 XIO B3:0/15 BND OTE O:0.0/3 EOR
%   B3:12/11  "Request to Send to Glaze or Repair" %
%   N7:12  "XFR4 STEP WORD" %
%   B3:1/1  "From Sealer Oven B TO Sanding Barn MODE" %
%   B3:0/15  "From Sanding Barn To TopCoat B MODE" %
%   O:0.0/3  SOL_XFR4_ROT  "Solenoid Transfer 4 Rotate" %
% Rung: 39 %
SOR END EOR

LADDER 4 "XFR 5"
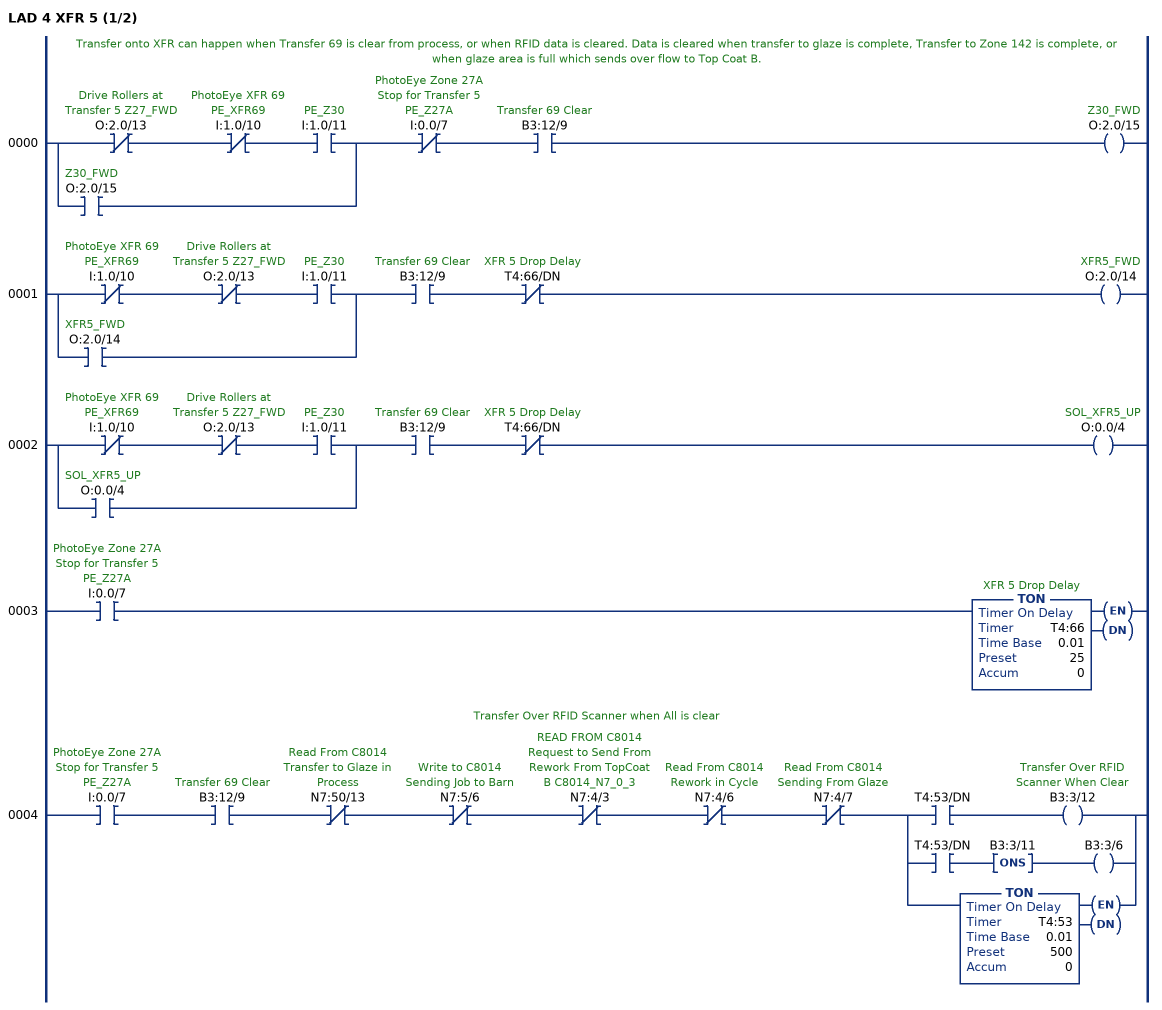
% Rung: 0 %
% Transfer onto XFR can happen when Transfer 69 is clear from process, or when RFID data is cleared. Data is cleared when transfer to glaze is complete, Transfer to Zone 142 is complete, or when glaze area is full which sends over flow to Top Coat B. %
SOR BST XIO O:2.0/13 XIO I:1.0/10 XIC I:1.0/11 NXB XIC O:2.0/15 BND XIO I:0.0/7 XIC B3:12/9 OTE O:2.0/15 EOR
%   O:2.0/13  Z27_FWD  "Drive Rollers at Transfer 5" %
%   I:1.0/10  PE_XFR69  "PhotoEye XFR 69" %
%   I:1.0/11  PE_Z30 %
%   O:2.0/15  Z30_FWD %
%   I:0.0/7  PE_Z27A  "PhotoEye Zone 27A Stop for Transfer 5" %
%   B3:12/9  "Transfer 69 Clear" %
% Rung: 1 %
SOR BST XIO I:1.0/10 XIO O:2.0/13 XIC I:1.0/11 NXB XIC O:2.0/14 BND XIC B3:12/9 XIO T4:66/DN OTE O:2.0/14 EOR
%   I:1.0/10  PE_XFR69  "PhotoEye XFR 69" %
%   O:2.0/13  Z27_FWD  "Drive Rollers at Transfer 5" %
%   I:1.0/11  PE_Z30 %
%   O:2.0/14  XFR5_FWD %
%   B3:12/9  "Transfer 69 Clear" %
%   T4:66  "XFR 5 Drop Delay" %
% Rung: 2 %
SOR BST XIO I:1.0/10 XIO O:2.0/13 XIC I:1.0/11 NXB XIC O:0.0/4 BND XIC B3:12/9 XIO T4:66/DN OTE O:0.0/4 EOR
%   I:1.0/10  PE_XFR69  "PhotoEye XFR 69" %
%   O:2.0/13  Z27_FWD  "Drive Rollers at Transfer 5" %
%   I:1.0/11  PE_Z30 %
%   O:0.0/4  SOL_XFR5_UP %
%   B3:12/9  "Transfer 69 Clear" %
%   T4:66  "XFR 5 Drop Delay" %
% Rung: 3 %
SOR XIC I:0.0/7 TON T4:66 0.01 25 0 EOR
%   I:0.0/7  PE_Z27A  "PhotoEye Zone 27A Stop for Transfer 5" %
%   T4:66  "XFR 5 Drop Delay" %
% Rung: 4 %
% Transfer Over RFID Scanner when All is clear %
SOR XIC I:0.0/7 XIC B3:12/9 XIO N7:50/13 XIO N7:5/6 XIO N7:4/3 XIO N7:4/6 XIO N7:4/7 BST XIC T4:53/DN OTE B3:3/12 NXB XIC T4:53/DN ONS B3:3/11 OTE B3:3/6 NXB TON T4:53 0.01 500 0 BND EOR
%   I:0.0/7  PE_Z27A  "PhotoEye Zone 27A Stop for Transfer 5" %
%   B3:12/9  "Transfer 69 Clear" %
%   N7:50/13  "Read From C8014 Transfer to Glaze in Process" %
%   N7:5/6  "Write to C8014 Sending Job to Barn" %
%   N7:4/3  C8014_N7_0_3  "READ FROM C8014 Request to Send From Rework From TopCoat B" %
%   N7:4/6  "Read From C8014 Rework in Cycle" %
%   N7:4/7  "Read From C8014 Sending From Glaze" %
%   B3:3/12  "Transfer Over RFID Scanner When Clear" %

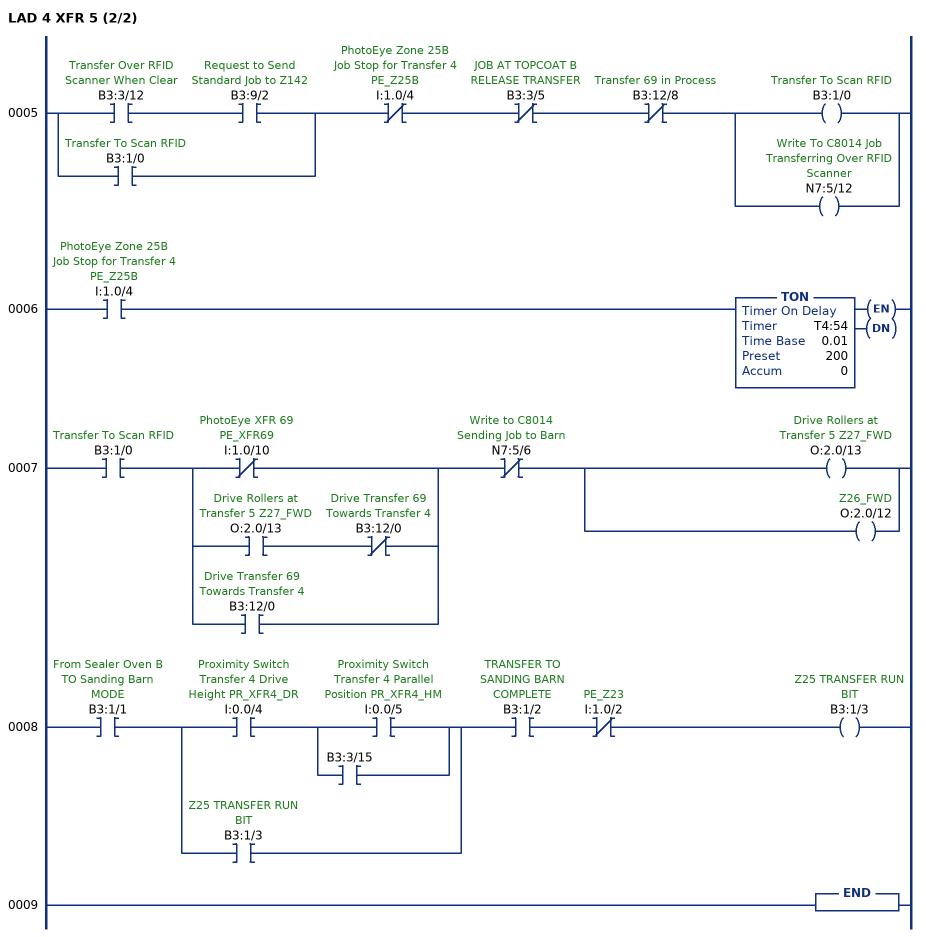
% Rung: 5 %
SOR BST XIC B3:3/12 XIC B3:9/2 NXB XIC B3:1/0 BND XIO I:1.0/4 XIO B3:3/5 XIO B3:12/8 BST OTE B3:1/0 NXB OTE N7:5/12 BND EOR
%   B3:3/12  "Transfer Over RFID Scanner When Clear" %
%   B3:9/2  "Request to Send Standard Job to Z142" %
%   B3:1/0  "Transfer To Scan RFID" %
%   I:1.0/4  PE_Z25B  "PhotoEye Zone 25B Job Stop for Transfer 4" %
%   B3:3/5  "JOB AT TOPCOAT B RELEASE TRANSFER" %
%   B3:12/8  "Transfer 69 in Process" %
%   N7:5/12  "Write To C8014 Job Transferring Over RFID Scanner" %
% Rung: 6 %
SOR XIC I:1.0/4 TON T4:54 0.01 200 0 EOR
%   I:1.0/4  PE_Z25B  "PhotoEye Zone 25B Job Stop for Transfer 4" %
% Rung: 7 %
SOR XIC B3:1/0 BST BST XIO I:1.0/10 NXB XIC O:2.0/13 XIO B3:12/0 BND NXB XIC B3:12/0 BND XIO N7:5/6 BST OTE O:2.0/13 NXB OTE O:2.0/12 BND EOR
%   B3:1/0  "Transfer To Scan RFID" %
%   I:1.0/10  PE_XFR69  "PhotoEye XFR 69" %
%   O:2.0/13  Z27_FWD  "Drive Rollers at Transfer 5" %
%   B3:12/0  "Drive Transfer 69 Towards Transfer 4" %
%   N7:5/6  "Write to C8014 Sending Job to Barn" %
%   O:2.0/12  Z26_FWD %
% Rung: 8 %
SOR XIC B3:1/1 BST XIC I:0.0/4 BST XIC I:0.0/5 NXB XIC B3:3/15 BND NXB XIC B3:1/3 BND XIC B3:1/2 XIO I:1.0/2 OTE B3:1/3 EOR
%   B3:1/1  "From Sealer Oven B TO Sanding Barn MODE" %
%   I:0.0/4  PR_XFR4_DR  "Proximity Switch Transfer 4 Drive Height" %
%   I:0.0/5  PR_XFR4_HM  "Proximity Switch Transfer 4 Parallel Position" %
%   B3:1/3  "Z25 TRANSFER RUN BIT" %
%   B3:1/2  "TRANSFER TO SANDING BARN COMPLETE" %
%   I:1.0/2  PE_Z23 %
% Rung: 9 %
SOR END EOR

LADDER 5 "XFR 6"
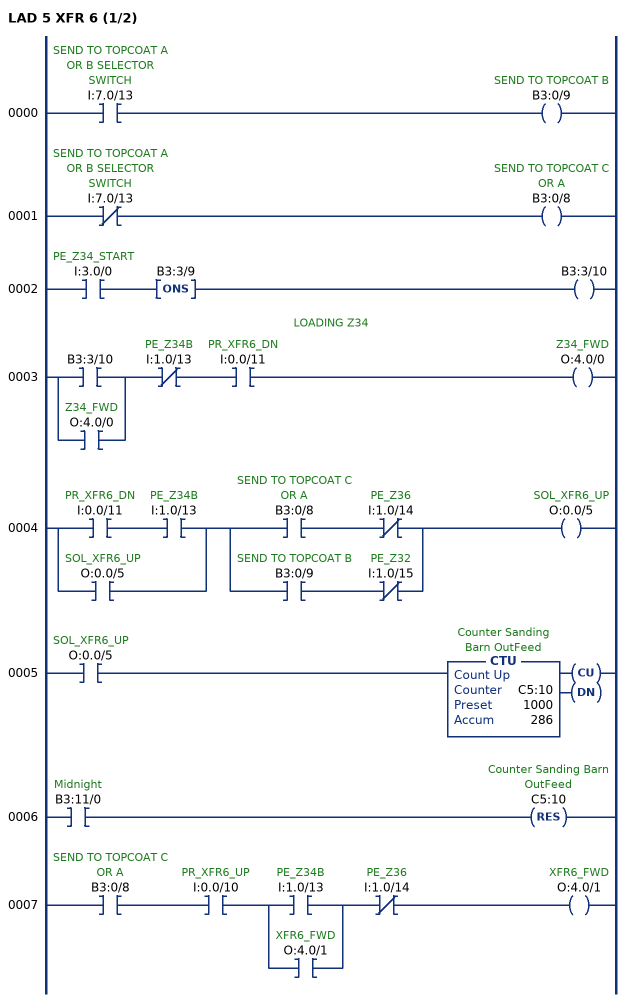
% Rung: 0 %
SOR XIC I:7.0/13 OTE B3:0/9 EOR
%   I:7.0/13  "SEND TO TOPCOAT A OR B SELECTOR SWITCH" %
%   B3:0/9  "SEND TO TOPCOAT B" %
% Rung: 1 %
SOR XIO I:7.0/13 OTE B3:0/8 EOR
%   I:7.0/13  "SEND TO TOPCOAT A OR B SELECTOR SWITCH" %
%   B3:0/8  "SEND TO TOPCOAT C OR A" %
% Rung: 2 %
SOR XIC I:3.0/0 ONS B3:3/9 OTE B3:3/10 EOR
%   I:3.0/0  PE_Z34_START %
% Rung: 3 %
% LOADING Z34 %
SOR BST XIC B3:3/10 NXB XIC O:4.0/0 BND XIO I:1.0/13 XIC I:0.0/11 OTE O:4.0/0 EOR
%   O:4.0/0  Z34_FWD %
%   I:1.0/13  PE_Z34B %
%   I:0.0/11  PR_XFR6_DN %
% Rung: 4 %
SOR BST XIC I:0.0/11 XIC I:1.0/13 NXB XIC O:0.0/5 BND BST XIC B3:0/8 XIO I:1.0/14 NXB XIC B3:0/9 XIO I:1.0/15 BND OTE O:0.0/5 EOR
%   I:0.0/11  PR_XFR6_DN %
%   I:1.0/13  PE_Z34B %
%   O:0.0/5  SOL_XFR6_UP %
%   B3:0/8  "SEND TO TOPCOAT C OR A" %
%   I:1.0/14  PE_Z36 %
%   B3:0/9  "SEND TO TOPCOAT B" %
%   I:1.0/15  PE_Z32 %
% Rung: 5 %
SOR XIC O:0.0/5 CTU C5:10 1000 286 EOR
%   O:0.0/5  SOL_XFR6_UP %
%   C5:10  "Counter Sanding Barn OutFeed" %
% Rung: 6 %
SOR XIC B3:11/0 RES C5:10 EOR
%   B3:11/0  "Midnight" %
%   C5:10  "Counter Sanding Barn OutFeed" %
% Rung: 7 %
SOR XIC B3:0/8 XIC I:0.0/10 BST XIC I:1.0/13 NXB XIC O:4.0/1 BND XIO I:1.0/14 OTE O:4.0/1 EOR
%   B3:0/8  "SEND TO TOPCOAT C OR A" %
%   I:0.0/10  PR_XFR6_UP %
%   I:1.0/13  PE_Z34B %
%   O:4.0/1  XFR6_FWD %
%   I:1.0/14  PE_Z36 %

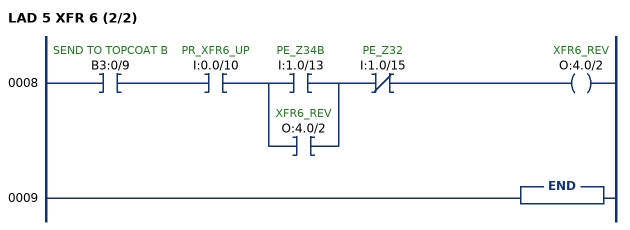
% Rung: 8 %
SOR XIC B3:0/9 XIC I:0.0/10 BST XIC I:1.0/13 NXB XIC O:4.0/2 BND XIO I:1.0/15 OTE O:4.0/2 EOR
%   B3:0/9  "SEND TO TOPCOAT B" %
%   I:0.0/10  PR_XFR6_UP %
%   I:1.0/13  PE_Z34B %
%   O:4.0/2  XFR6_REV %
%   I:1.0/15  PE_Z32 %
% Rung: 9 %
SOR END EOR

LADDER 6 "XFR 7"
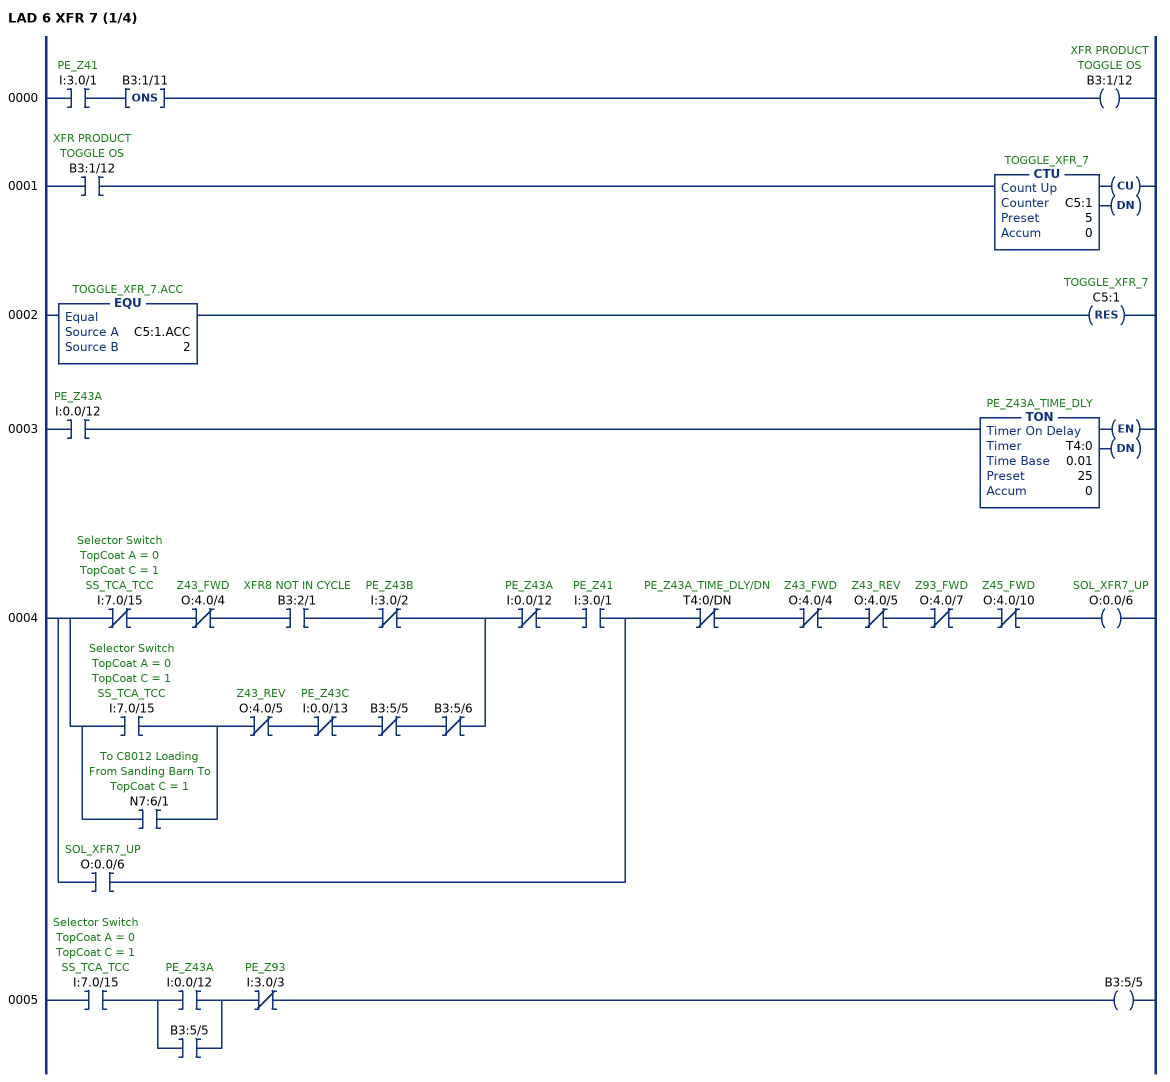
% Rung: 0 %
SOR XIC I:3.0/1 ONS B3:1/11 OTE B3:1/12 EOR
%   I:3.0/1  PE_Z41 %
%   B3:1/12  "XFR PRODUCT TOGGLE OS" %
% Rung: 1 %
SOR XIC B3:1/12 CTU C5:1 5 0 EOR
%   B3:1/12  "XFR PRODUCT TOGGLE OS" %
%   C5:1  TOGGLE_XFR_7 %
% Rung: 2 %
SOR EQU C5:1.ACC 2 RES C5:1 EOR
%   C5:1  TOGGLE_XFR_7 %
% Rung: 3 %
SOR XIC I:0.0/12 TON T4:0 0.01 25 0 EOR
%   I:0.0/12  PE_Z43A %
%   T4:0  PE_Z43A_TIME_DLY %
% Rung: 4 %
SOR BST BST XIO I:7.0/15 XIO O:4.0/4 XIC B3:2/1 XIO I:3.0/2 NXB BST XIC I:7.0/15 NXB XIC N7:6/1 BND XIO O:4.0/5 XIO I:0.0/13 XIO B3:5/5 XIO B3:5/6 BND XIO I:0.0/12 XIC I:3.0/1 NXB XIC O:0.0/6 BND XIO T4:0/DN XIO O:4.0/4 XIO O:4.0/5 XIO O:4.0/7 XIO O:4.0/10 OTE O:0.0/6 EOR
%   I:7.0/15  SS_TCA_TCC  "Selector Switch TopCoat A = 0 TopCoat C = 1" %
%   O:4.0/4  Z43_FWD %
%   B3:2/1  "XFR8 NOT IN CYCLE" %
%   I:3.0/2  PE_Z43B %
%   N7:6/1  "To C8012 Loading From Sanding Barn To TopCoat C = 1" %
%   O:4.0/5  Z43_REV %
%   I:0.0/13  PE_Z43C %
%   I:0.0/12  PE_Z43A %
%   I:3.0/1  PE_Z41 %
%   O:0.0/6  SOL_XFR7_UP %
%   T4:0  PE_Z43A_TIME_DLY %
%   O:4.0/7  Z93_FWD %
%   O:4.0/10  Z45_FWD %
% Rung: 5 %
SOR XIC I:7.0/15 BST XIC I:0.0/12 NXB XIC B3:5/5 BND XIO I:3.0/3 OTE B3:5/5 EOR
%   I:7.0/15  SS_TCA_TCC  "Selector Switch TopCoat A = 0 TopCoat C = 1" %
%   I:0.0/12  PE_Z43A %
%   I:3.0/3  PE_Z93 %

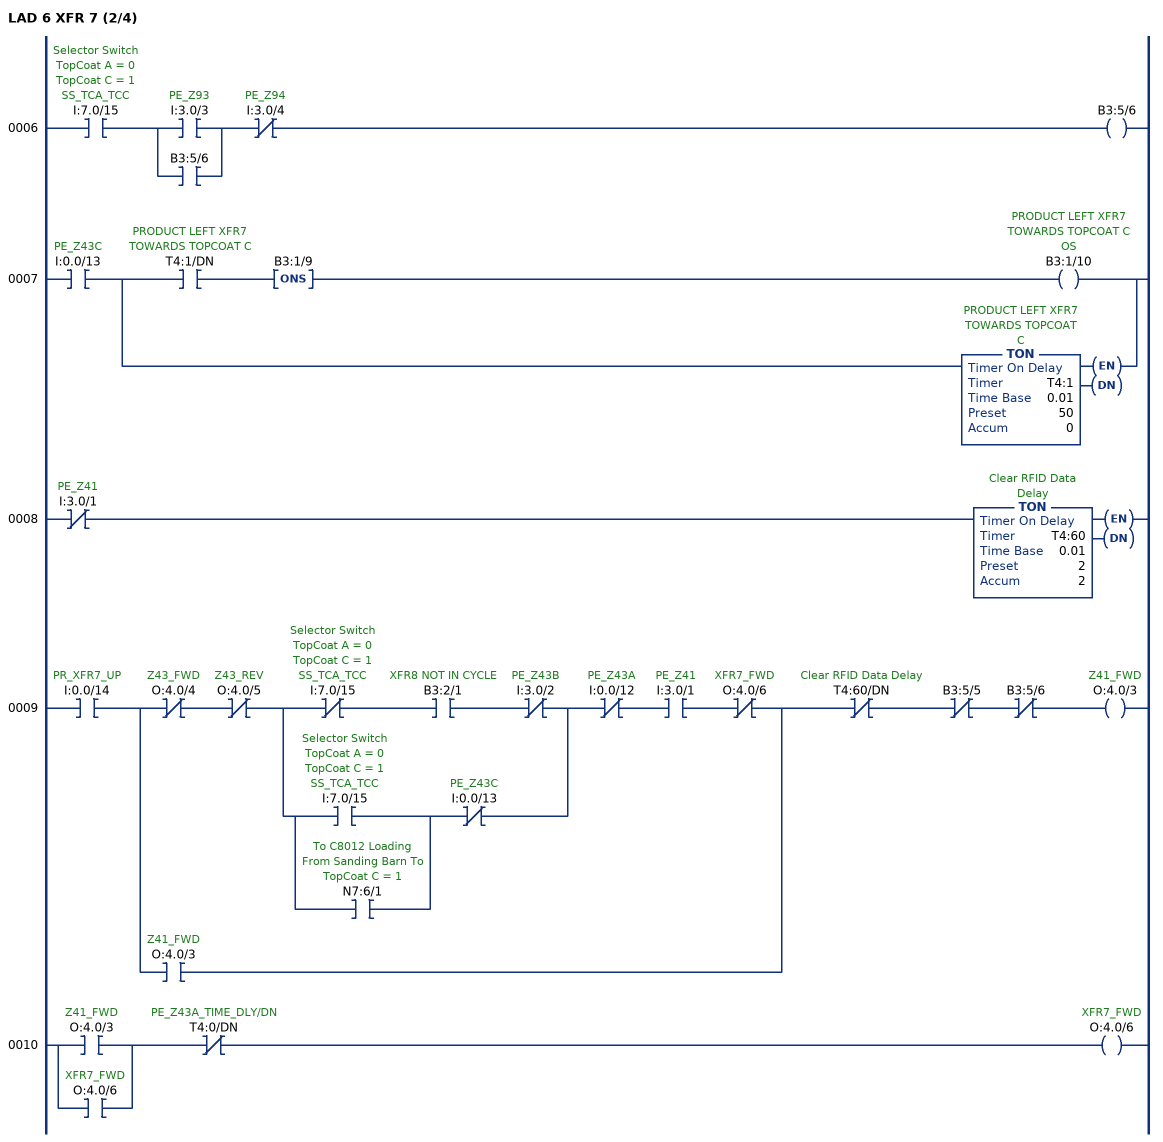
% Rung: 6 %
SOR XIC I:7.0/15 BST XIC I:3.0/3 NXB XIC B3:5/6 BND XIO I:3.0/4 OTE B3:5/6 EOR
%   I:7.0/15  SS_TCA_TCC  "Selector Switch TopCoat A = 0 TopCoat C = 1" %
%   I:3.0/3  PE_Z93 %
%   I:3.0/4  PE_Z94 %
% Rung: 7 %
SOR XIC I:0.0/13 BST XIC T4:1/DN ONS B3:1/9 OTE B3:1/10 NXB TON T4:1 0.01 50 0 BND EOR
%   I:0.0/13  PE_Z43C %
%   T4:1  "PRODUCT LEFT XFR7 TOWARDS TOPCOAT C" %
%   B3:1/10  "PRODUCT LEFT XFR7 TOWARDS TOPCOAT C OS" %
% Rung: 8 %
SOR XIO I:3.0/1 TON T4:60 0.01 2 2 EOR
%   I:3.0/1  PE_Z41 %
%   T4:60  "Clear RFID Data Delay" %
% Rung: 9 %
SOR XIC I:0.0/14 BST XIO O:4.0/4 XIO O:4.0/5 BST XIO I:7.0/15 XIC B3:2/1 XIO I:3.0/2 NXB BST XIC I:7.0/15 NXB XIC N7:6/1 BND XIO I:0.0/13 BND XIO I:0.0/12 XIC I:3.0/1 XIO O:4.0/6 NXB XIC O:4.0/3 BND XIO T4:60/DN XIO B3:5/5 XIO B3:5/6 OTE O:4.0/3 EOR
%   I:0.0/14  PR_XFR7_UP %
%   O:4.0/4  Z43_FWD %
%   O:4.0/5  Z43_REV %
%   I:7.0/15  SS_TCA_TCC  "Selector Switch TopCoat A = 0 TopCoat C = 1" %
%   B3:2/1  "XFR8 NOT IN CYCLE" %
%   I:3.0/2  PE_Z43B %
%   N7:6/1  "To C8012 Loading From Sanding Barn To TopCoat C = 1" %
%   I:0.0/13  PE_Z43C %
%   I:0.0/12  PE_Z43A %
%   I:3.0/1  PE_Z41 %
%   O:4.0/6  XFR7_FWD %
%   O:4.0/3  Z41_FWD %
%   T4:60  "Clear RFID Data Delay" %
% Rung: 10 %
SOR BST XIC O:4.0/3 NXB XIC O:4.0/6 BND XIO T4:0/DN OTE O:4.0/6 EOR
%   O:4.0/3  Z41_FWD %
%   O:4.0/6  XFR7_FWD %
%   T4:0  PE_Z43A_TIME_DLY %

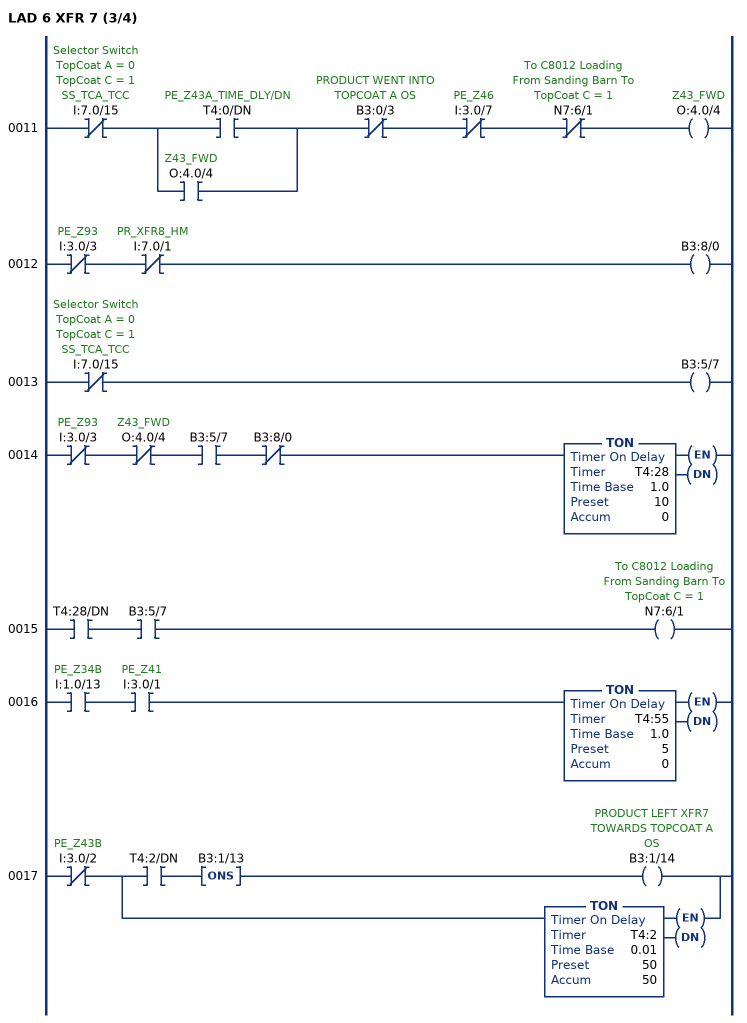
% Rung: 11 %
SOR XIO I:7.0/15 BST XIC T4:0/DN NXB XIC O:4.0/4 BND XIO B3:0/3 XIO I:3.0/7 XIO N7:6/1 OTE O:4.0/4 EOR
%   I:7.0/15  SS_TCA_TCC  "Selector Switch TopCoat A = 0 TopCoat C = 1" %
%   T4:0  PE_Z43A_TIME_DLY %
%   O:4.0/4  Z43_FWD %
%   B3:0/3  "PRODUCT WENT INTO TOPCOAT A OS" %
%   I:3.0/7  PE_Z46 %
%   N7:6/1  "To C8012 Loading From Sanding Barn To TopCoat C = 1" %
% Rung: 12 %
SOR XIO I:3.0/3 XIO I:7.0/1 OTE B3:8/0 EOR
%   I:3.0/3  PE_Z93 %
%   I:7.0/1  PR_XFR8_HM %
% Rung: 13 %
SOR XIO I:7.0/15 OTE B3:5/7 EOR
%   I:7.0/15  SS_TCA_TCC  "Selector Switch TopCoat A = 0 TopCoat C = 1" %
% Rung: 14 %
SOR XIO I:3.0/3 XIO O:4.0/4 XIC B3:5/7 XIO B3:8/0 TON T4:28 1.0 10 0 EOR
%   I:3.0/3  PE_Z93 %
%   O:4.0/4  Z43_FWD %
% Rung: 15 %
SOR XIC T4:28/DN XIC B3:5/7 OTE N7:6/1 EOR
%   N7:6/1  "To C8012 Loading From Sanding Barn To TopCoat C = 1" %
% Rung: 16 %
SOR XIC I:1.0/13 XIC I:3.0/1 TON T4:55 1.0 5 0 EOR
%   I:1.0/13  PE_Z34B %
%   I:3.0/1  PE_Z41 %
% Rung: 17 %
SOR XIO I:3.0/2 BST XIC T4:2/DN ONS B3:1/13 OTE B3:1/14 NXB TON T4:2 0.01 50 50 BND EOR
%   I:3.0/2  PE_Z43B %
%   B3:1/14  "PRODUCT LEFT XFR7 TOWARDS TOPCOAT A OS" %

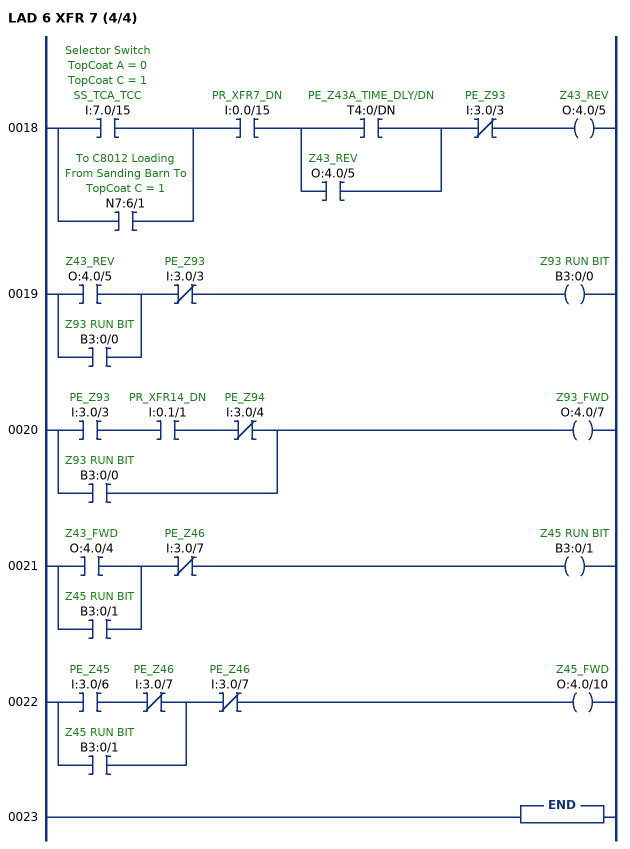
% Rung: 18 %
SOR BST XIC I:7.0/15 NXB XIC N7:6/1 BND XIC I:0.0/15 BST XIC T4:0/DN NXB XIC O:4.0/5 BND XIO I:3.0/3 OTE O:4.0/5 EOR
%   I:7.0/15  SS_TCA_TCC  "Selector Switch TopCoat A = 0 TopCoat C = 1" %
%   N7:6/1  "To C8012 Loading From Sanding Barn To TopCoat C = 1" %
%   I:0.0/15  PR_XFR7_DN %
%   T4:0  PE_Z43A_TIME_DLY %
%   O:4.0/5  Z43_REV %
%   I:3.0/3  PE_Z93 %
% Rung: 19 %
SOR BST XIC O:4.0/5 NXB XIC B3:0/0 BND XIO I:3.0/3 OTE B3:0/0 EOR
%   O:4.0/5  Z43_REV %
%   B3:0/0  "Z93 RUN BIT" %
%   I:3.0/3  PE_Z93 %
% Rung: 20 %
SOR BST XIC I:3.0/3 XIC I:0.1/1 XIO I:3.0/4 NXB XIC B3:0/0 BND OTE O:4.0/7 EOR
%   I:3.0/3  PE_Z93 %
%   I:0.1/1  PR_XFR14_DN %
%   I:3.0/4  PE_Z94 %
%   B3:0/0  "Z93 RUN BIT" %
%   O:4.0/7  Z93_FWD %
% Rung: 21 %
SOR BST XIC O:4.0/4 NXB XIC B3:0/1 BND XIO I:3.0/7 OTE B3:0/1 EOR
%   O:4.0/4  Z43_FWD %
%   B3:0/1  "Z45 RUN BIT" %
%   I:3.0/7  PE_Z46 %
% Rung: 22 %
SOR BST XIC I:3.0/6 XIO I:3.0/7 NXB XIC B3:0/1 BND XIO I:3.0/7 OTE O:4.0/10 EOR
%   I:3.0/6  PE_Z45 %
%   I:3.0/7  PE_Z46 %
%   B3:0/1  "Z45 RUN BIT" %
%   O:4.0/10  Z45_FWD %
% Rung: 23 %
SOR END EOR

LADDER 7 "XFR 8"
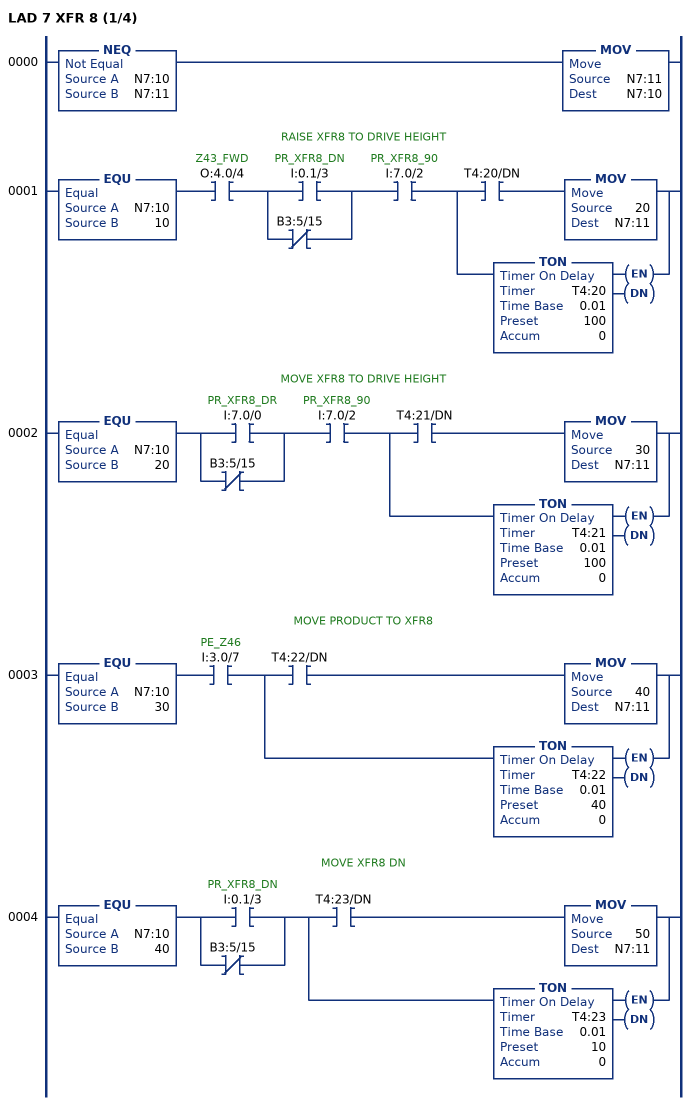
% Rung: 0 %
SOR NEQ N7:10 N7:11 MOV N7:11 N7:10 EOR
% Rung: 1 %
% RAISE XFR8 TO DRIVE HEIGHT %
SOR EQU N7:10 10 XIC O:4.0/4 BST XIC I:0.1/3 NXB XIO B3:5/15 BND XIC I:7.0/2 BST XIC T4:20/DN MOV 20 N7:11 NXB TON T4:20 0.01 100 0 BND EOR
%   O:4.0/4  Z43_FWD %
%   I:0.1/3  PR_XFR8_DN %
%   I:7.0/2  PR_XFR8_90 %
% Rung: 2 %
% MOVE XFR8 TO DRIVE HEIGHT %
SOR EQU N7:10 20 BST XIC I:7.0/0 NXB XIO B3:5/15 BND XIC I:7.0/2 BST XIC T4:21/DN MOV 30 N7:11 NXB TON T4:21 0.01 100 0 BND EOR
%   I:7.0/0  PR_XFR8_DR %
%   I:7.0/2  PR_XFR8_90 %
% Rung: 3 %
% MOVE PRODUCT TO XFR8 %
SOR EQU N7:10 30 XIC I:3.0/7 BST XIC T4:22/DN MOV 40 N7:11 NXB TON T4:22 0.01 40 0 BND EOR
%   I:3.0/7  PE_Z46 %
% Rung: 4 %
% MOVE XFR8 DN %
SOR EQU N7:10 40 BST XIC I:0.1/3 NXB XIO B3:5/15 BND BST XIC T4:23/DN MOV 50 N7:11 NXB TON T4:23 0.01 10 0 BND EOR
%   I:0.1/3  PR_XFR8_DN %

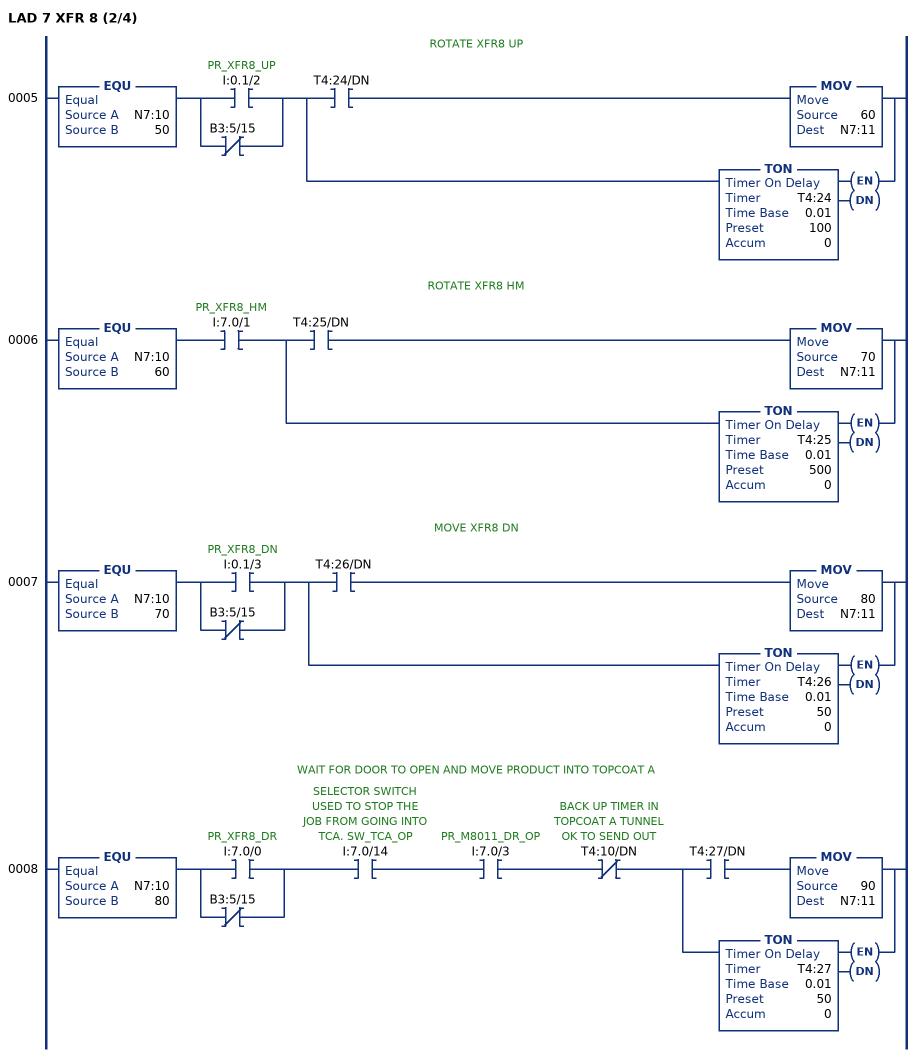
% Rung: 5 %
% ROTATE XFR8 UP %
SOR EQU N7:10 50 BST XIC I:0.1/2 NXB XIO B3:5/15 BND BST XIC T4:24/DN MOV 60 N7:11 NXB TON T4:24 0.01 100 0 BND EOR
%   I:0.1/2  PR_XFR8_UP %
% Rung: 6 %
% ROTATE XFR8 HM %
SOR EQU N7:10 60 XIC I:7.0/1 BST XIC T4:25/DN MOV 70 N7:11 NXB TON T4:25 0.01 500 0 BND EOR
%   I:7.0/1  PR_XFR8_HM %
% Rung: 7 %
% MOVE XFR8 DN %
SOR EQU N7:10 70 BST XIC I:0.1/3 NXB XIO B3:5/15 BND BST XIC T4:26/DN MOV 80 N7:11 NXB TON T4:26 0.01 50 0 BND EOR
%   I:0.1/3  PR_XFR8_DN %
% Rung: 8 %
% WAIT FOR DOOR TO OPEN AND MOVE PRODUCT INTO TOPCOAT A %
SOR EQU N7:10 80 BST XIC I:7.0/0 NXB XIO B3:5/15 BND XIC I:7.0/14 XIC I:7.0/3 XIO T4:10/DN BST XIC T4:27/DN MOV 90 N7:11 NXB TON T4:27 0.01 50 0 BND EOR
%   I:7.0/0  PR_XFR8_DR %
%   I:7.0/14  SW_TCA_OP  "SELECTOR SWITCH USED TO STOP THE JOB FROM GOING INTO TCA." %
%   I:7.0/3  PR_M8011_DR_OP %
%   T4:10  "BACK UP TIMER IN TOPCOAT A TUNNEL OK TO SEND OUT" %

